Yaskawa INFORM job: A_ROOF_UPPER_0614_2_PAINT_56.JBI

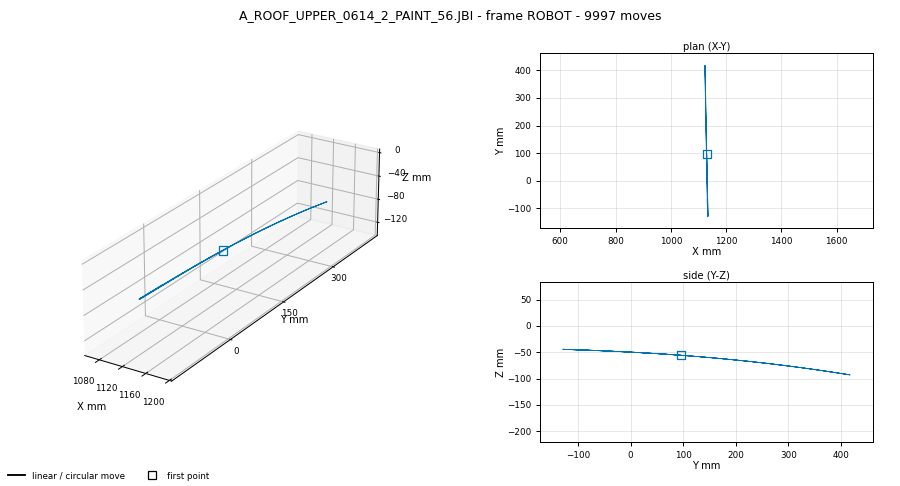
[picture p0: tool path of A_ROOF_UPPER_0614_2_PAINT_56.JBI in frame ROBOT, 9997 of 9997 moves have a stored position in this frame; points joined in program order, loops and branches not executed]
/JOB
//NAME A_ROOF_UPPER_0614_2_PAINT56
//POS
///NPOS 9997,0,0,0,0,0
///TOOL 1
///USER 0
///POSTYPE ROBOT
///RECTAN
///RCONF 1,0,0,0,0,0,0,0,0,0,0,0,0,0,0,0,0,0,0,0,0,0,0,0
C00000=1130.429,96.050,-55.597,-179.993,7.913,149.501
C00001=1130.433,95.801,-55.579,-179.995,7.908,149.501
C00002=1130.438,95.552,-55.561,-179.997,7.904,149.500
C00003=1130.443,95.303,-55.543,-179.999,7.901,149.500
C00004=1130.448,95.054,-55.525,180.000,7.897,149.500
C00005=1130.453,94.805,-55.507,179.998,7.893,149.499
C00006=1130.457,94.555,-55.488,179.996,7.888,149.499
C00007=1130.463,94.305,-55.470,179.994,7.884,149.499
C00008=1130.468,94.056,-55.452,179.993,7.881,149.498
C00009=1130.473,93.807,-55.434,179.991,7.877,149.498
C00010=1130.478,93.558,-55.416,179.989,7.873,149.497
C00011=1130.483,93.308,-55.398,179.987,7.869,149.497
C00012=1130.488,93.059,-55.380,179.986,7.865,149.497
C00013=1130.493,92.810,-55.362,179.984,7.861,149.496
C00014=1130.497,92.560,-55.344,179.982,7.857,149.496
C00015=1130.502,92.311,-55.326,179.980,7.853,149.495
C00016=1130.507,92.062,-55.308,179.979,7.849,149.495
C00017=1130.512,91.813,-55.290,179.977,7.845,149.495
C00018=1130.517,91.564,-55.272,179.976,7.841,149.494
C00019=1130.521,91.314,-55.254,179.974,7.837,149.494
C00020=1130.526,91.065,-55.236,179.972,7.833,149.493
C00021=1130.532,90.815,-55.218,179.971,7.830,149.493
C00022=1130.536,90.566,-55.200,179.970,7.825,149.492
C00023=1130.541,90.317,-55.182,179.968,7.821,149.492
C00024=1130.545,90.102,-55.167,179.967,7.819,149.492
C00025=1130.549,89.887,-55.151,179.965,7.815,149.491
C00026=1130.553,89.672,-55.137,179.964,7.812,149.491
C00027=1130.558,89.457,-55.121,179.963,7.808,149.490
C00028=1130.562,89.242,-55.105,179.962,7.805,149.490
C00029=1130.567,89.027,-55.090,179.960,7.801,149.489
C00030=1130.570,88.811,-55.075,179.959,7.798,149.489
C00031=1130.575,88.596,-55.060,179.958,7.795,149.489
C00032=1130.579,88.347,-55.042,179.956,7.791,149.488
C00033=1130.585,88.097,-55.024,179.955,7.787,149.488
C00034=1130.590,87.848,-55.006,179.953,7.783,149.487
C00035=1130.594,87.599,-54.989,179.952,7.779,149.487
C00036=1130.599,87.350,-54.971,179.950,7.775,149.486
C00037=1130.604,87.100,-54.954,179.949,7.771,149.486
C00038=1130.609,86.851,-54.936,179.947,7.767,149.485
C00039=1130.614,86.602,-54.918,179.946,7.764,149.485
C00040=1130.619,86.352,-54.900,179.945,7.760,149.485
C00041=1130.623,86.103,-54.883,179.944,7.756,149.484
C00042=1130.628,85.854,-54.865,179.942,7.752,149.483
C00043=1130.633,85.604,-54.848,179.940,7.748,149.483
C00044=1130.638,85.355,-54.830,179.939,7.744,149.483
C00045=1130.643,85.105,-54.813,179.938,7.740,149.482
C00046=1130.648,84.856,-54.795,179.937,7.737,149.482
C00047=1130.653,84.608,-54.778,179.935,7.733,149.481
C00048=1130.658,84.358,-54.760,179.934,7.728,149.480
C00049=1130.663,84.109,-54.742,179.933,7.725,149.480
C00050=1130.668,83.859,-54.725,179.931,7.721,149.480
C00051=1130.673,83.610,-54.708,179.930,7.717,149.479
C00052=1130.678,83.361,-54.690,179.929,7.713,149.479
C00053=1130.683,83.111,-54.672,179.928,7.710,149.478
C00054=1130.688,82.862,-54.655,179.927,7.706,149.477
C00055=1130.692,82.613,-54.638,179.925,7.702,149.477
C00056=1130.697,82.363,-54.621,179.925,7.698,149.476
C00057=1130.702,82.114,-54.603,179.923,7.694,149.476
C00058=1130.707,81.864,-54.586,179.922,7.690,149.475
C00059=1130.712,81.615,-54.568,179.921,7.687,149.475
C00060=1130.717,81.366,-54.551,179.920,7.683,149.474
C00061=1130.722,81.117,-54.534,179.919,7.680,149.474
C00062=1130.727,80.867,-54.516,179.918,7.675,149.473
C00063=1130.732,80.618,-54.499,179.916,7.672,149.473
C00064=1130.736,80.369,-54.482,179.916,7.668,149.472
C00065=1130.741,80.119,-54.464,179.914,7.664,149.472
C00066=1130.746,79.870,-54.446,179.913,7.661,149.471
C00067=1130.751,79.620,-54.430,179.912,7.657,149.471
C00068=1130.757,79.371,-54.413,179.911,7.653,149.470
C00069=1130.762,79.122,-54.395,179.910,7.649,149.470
C00070=1130.766,78.872,-54.378,179.909,7.645,149.469
C00071=1130.771,78.623,-54.361,179.908,7.642,149.469
C00072=1130.776,78.373,-54.343,179.907,7.638,149.468
C00073=1130.781,78.124,-54.326,179.906,7.634,149.467
C00074=1130.786,77.874,-54.309,179.905,7.631,149.467
C00075=1130.791,77.626,-54.292,179.903,7.627,149.466
C00076=1130.796,77.376,-54.275,179.903,7.624,149.466
C00077=1130.801,77.126,-54.257,179.902,7.619,149.465
C00078=1130.805,76.878,-54.240,179.901,7.616,149.465
C00079=1130.810,76.628,-54.223,179.900,7.612,149.464
C00080=1130.819,76.209,-54.195,179.897,7.606,149.463
C00081=1130.827,75.790,-54.166,179.895,7.599,149.463
C00082=1130.835,75.371,-54.137,179.892,7.592,149.462
C00083=1130.844,74.952,-54.108,179.890,7.586,149.461
C00084=1130.849,74.703,-54.092,179.889,7.582,149.460
C00085=1130.854,74.454,-54.074,179.887,7.578,149.460
C00086=1130.858,74.204,-54.057,179.886,7.574,149.460
C00087=1130.863,73.954,-54.040,179.885,7.570,149.459
C00088=1130.868,73.705,-54.023,179.883,7.566,149.458
C00089=1130.873,73.456,-54.007,179.881,7.562,149.458
C00090=1130.878,73.206,-53.990,179.880,7.558,149.458
C00091=1130.883,72.957,-53.973,179.879,7.554,149.457
C00092=1130.888,72.707,-53.956,179.877,7.550,149.457
C00093=1130.893,72.459,-53.939,179.876,7.546,149.456
C00094=1130.898,72.209,-53.922,179.874,7.542,149.456
C00095=1130.902,71.960,-53.905,179.873,7.538,149.455
C00096=1130.908,71.711,-53.888,179.871,7.534,149.455
C00097=1130.913,71.461,-53.871,179.870,7.530,149.454
C00098=1130.917,71.212,-53.855,179.868,7.526,149.454
C00099=1130.922,70.962,-53.837,179.867,7.522,149.453
C00100=1130.928,70.713,-53.821,179.865,7.518,149.453
C00101=1130.933,70.463,-53.804,179.864,7.514,149.452
C00102=1130.937,70.214,-53.787,179.862,7.510,149.452
C00103=1130.942,69.965,-53.771,179.861,7.506,149.451
C00104=1130.968,68.716,-53.685,-179.718,6.654,149.139
C00105=1130.972,68.467,-53.668,-179.720,6.653,149.139
C00106=1130.977,68.217,-53.652,-179.723,6.652,149.139
C00107=1130.982,67.969,-53.636,-179.726,6.650,149.140
C00108=1130.986,67.718,-53.620,-179.728,6.648,149.140
C00109=1130.992,67.469,-53.603,-179.731,6.648,149.141
C00110=1130.997,67.220,-53.586,-179.734,6.646,149.141
C00111=1131.002,66.970,-53.570,-179.736,6.645,149.142
C00112=1131.007,66.721,-53.554,-179.739,6.643,149.142
C00113=1131.011,66.471,-53.537,-179.741,6.642,149.143
C00114=1131.017,66.222,-53.521,-179.745,6.641,149.143
C00115=1131.022,65.972,-53.504,-179.747,6.639,149.144
C00116=1131.027,65.724,-53.488,-179.750,6.638,149.144
C00117=1131.032,65.473,-53.472,-179.752,6.637,149.145
C00118=1131.037,65.225,-53.456,-179.756,6.636,149.145
C00119=1131.041,64.975,-53.439,-179.758,6.634,149.146
C00120=1131.047,64.726,-53.423,-179.760,6.633,149.146
C00121=1131.051,64.476,-53.407,-179.763,6.631,149.147
C00122=1131.056,64.227,-53.391,-179.766,6.630,149.147
C00123=1131.061,63.977,-53.374,-179.769,6.629,149.148
C00124=1131.066,63.728,-53.359,-179.771,6.628,149.148
C00125=1131.071,63.478,-53.342,-179.774,6.626,149.149
C00126=1131.077,63.229,-53.325,-179.777,6.624,149.149
C00127=1131.081,62.979,-53.309,-179.779,6.624,149.150
C00128=1131.086,62.730,-53.293,-179.782,6.622,149.150
C00129=1131.091,62.480,-53.277,-179.785,6.621,149.151
C00130=1131.096,62.232,-53.261,-179.787,6.620,149.151
C00131=1131.101,61.981,-53.245,-179.790,6.619,149.152
C00132=1131.106,61.733,-53.229,-179.793,6.617,149.152
C00133=1131.112,61.483,-53.213,-179.795,6.616,149.153
C00134=1131.116,61.234,-53.196,-179.798,6.614,149.153
C00135=1131.121,60.984,-53.181,-179.801,6.613,149.154
C00136=1131.126,60.734,-53.165,-179.803,6.612,149.154
C00137=1131.131,60.486,-53.148,-179.806,6.611,149.155
C00138=1131.136,60.235,-53.133,-179.809,6.609,149.155
C00139=1131.141,59.987,-53.116,-179.811,6.608,149.155
C00140=1131.147,59.737,-53.101,-179.814,6.607,149.156
C00141=1131.151,59.487,-53.085,-179.817,6.605,149.157
C00142=1131.156,59.238,-53.068,-179.819,6.605,149.157
C00143=1131.161,58.988,-53.052,-179.822,6.603,149.157
C00144=1131.166,58.739,-53.036,-179.825,6.602,149.158
C00145=1131.172,58.490,-53.021,-179.827,6.601,149.159
C00146=1131.176,58.240,-53.005,-179.830,6.599,149.159
C00147=1131.181,57.992,-52.989,-179.833,6.598,149.159
C00148=1131.186,57.741,-52.973,-179.836,6.597,149.160
C00149=1131.191,57.492,-52.957,-179.838,6.595,149.161
C00150=1131.196,57.243,-52.942,-179.841,6.594,149.161
C00151=1131.201,56.993,-52.925,-179.843,6.593,149.161
C00152=1131.206,56.744,-52.909,-179.847,6.592,149.162
C00153=1131.212,56.494,-52.894,-179.849,6.590,149.163
C00154=1131.216,56.245,-52.877,-179.851,6.589,149.163
C00155=1131.221,55.995,-52.862,-179.854,6.588,149.163
C00156=1131.226,55.746,-52.847,-179.857,6.586,149.164
C00157=1131.231,55.496,-52.831,-179.860,6.586,149.165
C00158=1131.236,55.247,-52.815,-179.862,6.584,149.165
C00159=1131.241,54.998,-52.799,-179.865,6.582,149.165
C00160=1131.246,54.748,-52.783,-179.868,6.582,149.166
C00161=1131.252,54.499,-52.767,-179.870,6.580,149.167
C00162=1131.256,54.249,-52.752,-179.873,6.579,149.167
C00163=1131.261,53.999,-52.736,-179.875,6.578,149.167
C00164=1131.266,53.751,-52.720,-179.879,6.576,149.168
C00165=1131.272,53.481,-52.704,-179.881,6.575,149.168
C00166=1131.277,53.213,-52.687,-179.884,6.574,149.169
C00167=1131.283,52.944,-52.670,-179.887,6.573,149.170
C00168=1131.289,52.676,-52.653,-179.890,6.571,149.170
C00169=1131.293,52.426,-52.637,-179.893,6.570,149.171
C00170=1131.298,52.177,-52.622,-179.895,6.569,149.171
C00171=1131.303,51.927,-52.606,-179.898,6.567,149.172
C00172=1131.308,51.677,-52.590,-179.901,6.566,149.172
C00173=1131.313,51.428,-52.575,-179.903,6.565,149.173
C00174=1131.318,51.179,-52.560,-179.906,6.564,149.173
C00175=1131.324,50.929,-52.544,-179.908,6.563,149.174
C00176=1131.328,50.680,-52.529,-179.911,6.562,149.174
C00177=1131.333,50.430,-52.513,-179.914,6.560,149.175
C00178=1131.338,50.181,-52.497,-179.916,6.559,149.175
C00179=1131.344,49.932,-52.481,-179.919,6.557,149.176
C00180=1131.348,49.682,-52.466,-179.922,6.557,149.176
C00181=1131.353,49.433,-52.450,-179.924,6.555,149.177
C00182=1131.359,49.183,-52.435,-179.927,6.554,149.177
C00183=1131.363,48.934,-52.420,-179.929,6.553,149.178
C00184=1131.369,48.684,-52.405,-179.933,6.552,149.178
C00185=1131.373,48.434,-52.389,-179.935,6.551,149.179
C00186=1131.378,48.185,-52.374,-179.937,6.549,149.179
C00187=1131.384,47.936,-52.358,-179.941,6.548,149.180
C00188=1131.388,47.687,-52.343,-179.943,6.547,149.180
C00189=1131.394,47.437,-52.328,-179.946,6.546,149.181
C00190=1131.398,47.187,-52.312,-179.948,6.545,149.181
C00191=1131.403,46.938,-52.297,-179.951,6.543,149.182
C00192=1131.408,46.689,-52.281,-179.953,6.543,149.182
C00193=1131.414,46.439,-52.266,-179.956,6.541,149.183
C00194=1131.419,46.190,-52.251,-179.959,6.539,149.183
C00195=1131.424,45.939,-52.235,-179.961,6.539,149.184
C00196=1131.428,45.690,-52.220,-179.964,6.537,149.184
C00197=1131.434,45.441,-52.205,-179.966,6.536,149.185
C00198=1131.438,45.192,-52.190,-179.970,6.535,149.185
C00199=1131.444,44.942,-52.174,-179.972,6.534,149.186
C00200=1131.449,44.692,-52.159,-179.974,6.533,149.186
C00201=1131.454,44.443,-52.144,-179.977,6.531,149.187
C00202=1131.459,44.193,-52.128,-179.980,6.531,149.187
C00203=1131.463,43.944,-52.113,-179.983,6.529,149.188
C00204=1131.469,43.695,-52.098,-179.985,6.528,149.188
C00205=1131.474,43.445,-52.083,-179.988,6.527,149.189
C00206=1131.479,43.196,-52.068,-179.990,6.526,149.189
C00207=1131.484,42.947,-52.053,-179.993,6.525,149.190
C00208=1131.489,42.697,-52.038,-179.995,6.524,149.190
C00209=1131.494,42.447,-52.023,-179.998,6.522,149.191
C00210=1131.499,42.198,-52.007,179.999,6.522,149.191
C00211=1131.504,41.949,-51.992,179.997,6.520,149.192
C00212=1131.509,41.698,-51.977,179.994,6.518,149.192
C00213=1131.514,41.449,-51.962,179.991,6.518,149.193
C00214=1131.519,41.200,-51.947,179.989,6.516,149.193
C00215=1131.524,40.950,-51.932,179.986,6.516,149.194
C00216=1131.530,40.701,-51.917,179.983,6.514,149.195
C00217=1131.534,40.452,-51.902,179.981,6.513,149.195
C00218=1131.539,40.202,-51.887,179.978,6.512,149.196
C00219=1131.545,39.952,-51.872,179.976,6.511,149.196
C00220=1131.550,39.703,-51.858,179.973,6.510,149.197
C00221=1131.555,39.453,-51.842,179.971,6.509,149.197
C00222=1131.560,39.204,-51.827,179.968,6.507,149.198
C00223=1131.565,38.954,-51.813,179.965,6.507,149.198
C00224=1131.570,38.705,-51.797,179.962,6.505,149.199
C00225=1131.575,38.455,-51.783,179.960,6.504,149.199
C00226=1131.580,38.206,-51.767,179.957,6.503,149.200
C00227=1131.585,37.956,-51.753,179.955,6.502,149.200
C00228=1131.590,37.707,-51.738,179.952,6.501,149.201
C00229=1131.596,37.457,-51.723,179.950,6.500,149.201
C00230=1131.600,37.208,-51.708,179.947,6.499,149.202
C00231=1131.606,36.958,-51.693,179.945,6.498,149.202
C00232=1131.611,36.709,-51.678,179.942,6.496,149.203
C00233=1131.615,36.459,-51.664,179.939,6.496,149.203
C00234=1131.621,36.210,-51.648,179.936,6.494,149.204
C00235=1131.626,35.960,-51.634,179.934,6.493,149.204
C00236=1131.630,35.711,-51.619,179.931,6.492,149.205
C00237=1131.636,35.461,-51.604,179.929,6.491,149.205
C00238=1131.641,35.212,-51.589,179.926,6.490,149.206
C00239=1131.646,34.962,-51.575,179.924,6.489,149.206
C00240=1131.650,34.713,-51.560,179.921,6.488,149.207
C00241=1131.656,34.463,-51.545,179.918,6.487,149.207
C00242=1131.661,34.213,-51.531,179.916,6.485,149.208
C00243=1131.666,33.964,-51.516,179.913,6.485,149.209
C00244=1131.671,33.715,-51.502,179.910,6.483,149.209
C00245=1131.676,33.465,-51.487,179.908,6.482,149.209
C00246=1131.681,33.215,-51.472,179.905,6.481,149.210
C00247=1131.686,32.966,-51.457,179.903,6.480,149.211
C00248=1131.691,32.716,-51.443,179.900,6.479,149.211
C00249=1131.697,32.467,-51.428,179.898,6.478,149.212
C00250=1131.702,32.218,-51.414,179.894,6.477,149.212
C00251=1131.707,31.968,-51.399,179.892,6.476,149.213
C00252=1131.711,31.719,-51.384,179.890,6.474,149.213
C00253=1131.717,31.469,-51.370,179.887,6.474,149.214
C00254=1131.722,31.219,-51.355,179.884,6.472,149.214
C00255=1131.727,30.970,-51.340,179.882,6.471,149.215
C00256=1131.732,30.720,-51.326,179.879,6.470,149.215
C00257=1131.737,30.471,-51.312,179.877,6.469,149.216
C00258=1131.742,30.221,-51.297,179.874,6.468,149.216
C00259=1131.748,29.972,-51.282,179.872,6.467,149.217
C00260=1131.753,29.722,-51.268,179.869,6.466,149.217
C00261=1131.758,29.473,-51.254,179.866,6.465,149.218
C00262=1131.762,29.223,-51.239,179.864,6.464,149.218
C00263=1131.767,28.973,-51.225,179.861,6.463,149.219
C00264=1131.772,28.724,-51.210,179.859,6.462,149.219
C00265=1131.777,28.475,-51.196,179.856,6.460,149.220
C00266=1131.783,28.225,-51.181,179.854,6.459,149.220
C00267=1131.788,27.975,-51.167,179.851,6.459,149.221
C00268=1131.793,27.726,-51.153,179.848,6.457,149.221
C00269=1131.798,27.457,-51.137,179.845,6.456,149.222
C00270=1131.804,27.188,-51.121,179.843,6.455,149.223
C00271=1131.809,26.919,-51.106,179.840,6.454,149.223
C00272=1131.815,26.650,-51.090,179.837,6.453,149.224
C00273=1131.820,26.401,-51.076,179.835,6.452,149.224
C00274=1131.825,26.151,-51.062,179.832,6.451,149.225
C00275=1131.830,25.901,-51.048,179.829,6.450,149.225
C00276=1131.835,25.652,-51.033,179.827,6.449,149.226
C00277=1131.840,25.402,-51.019,179.824,6.448,149.226
C00278=1131.846,25.153,-51.005,179.822,6.447,149.227
C00279=1131.851,24.903,-50.991,179.819,6.446,149.227
C00280=1131.856,24.653,-50.977,179.816,6.445,149.228
C00281=1131.861,24.404,-50.962,179.814,6.444,149.229
C00282=1131.866,24.155,-50.948,179.811,6.442,149.229
C00283=1131.871,23.905,-50.934,179.809,6.441,149.229
C00284=1131.876,23.655,-50.920,179.806,6.441,149.230
C00285=1131.881,23.406,-50.906,179.804,6.439,149.231
C00286=1131.886,23.156,-50.891,179.801,6.439,149.231
C00287=1131.892,22.907,-50.877,179.798,6.437,149.232
C00288=1131.896,22.657,-50.863,179.796,6.437,149.232
C00289=1131.901,22.407,-50.849,179.794,6.436,149.233
C00290=1131.906,22.158,-50.835,179.791,6.434,149.233
C00291=1131.912,21.909,-50.821,179.788,6.434,149.234
C00292=1131.917,21.659,-50.806,179.786,6.432,149.234
C00293=1131.922,21.409,-50.792,179.783,6.432,149.235
C00294=1131.927,21.160,-50.778,179.781,6.431,149.235
C00295=1131.932,20.911,-50.764,179.778,6.429,149.236
C00296=1131.937,20.661,-50.750,179.775,6.429,149.237
C00297=1131.942,20.411,-50.737,179.773,6.427,149.237
C00298=1131.947,20.162,-50.723,179.771,6.426,149.237
C00299=1131.952,19.912,-50.708,179.768,6.426,149.238
C00300=1131.957,19.662,-50.694,179.765,6.424,149.239
C00301=1131.963,19.413,-50.680,179.763,6.423,149.239
C00302=1131.968,19.164,-50.666,179.760,6.422,149.239
C00303=1131.973,18.914,-50.652,179.757,6.421,149.240
C00304=1131.979,18.664,-50.639,179.755,6.421,149.241
C00305=1131.983,18.415,-50.625,179.753,6.419,149.241
C00306=1131.988,18.165,-50.611,179.750,6.419,149.242
C00307=1131.993,17.916,-50.597,179.748,6.418,149.242
C00308=1131.998,17.666,-50.582,179.745,6.416,149.243
C00309=1132.004,17.416,-50.569,179.742,6.416,149.243
C00310=1132.009,17.167,-50.555,179.740,6.415,149.244
C00311=1132.013,16.918,-50.541,179.737,6.413,149.244
C00312=1132.018,16.668,-50.527,179.735,6.413,149.245
C00313=1132.024,16.418,-50.514,179.732,6.411,149.245
C00314=1132.029,16.169,-50.499,179.730,6.411,149.246
C00315=1132.034,15.919,-50.485,179.727,6.410,149.247
C00316=1132.039,15.670,-50.473,179.724,6.408,149.247
C00317=1132.044,15.420,-50.458,179.722,6.408,149.248
C00318=1132.049,15.170,-50.444,179.719,6.407,149.248
C00319=1132.055,14.921,-50.430,179.717,6.406,149.249
C00320=1132.060,14.671,-50.417,179.715,6.405,149.249
C00321=1132.065,14.422,-50.403,179.712,6.404,149.250
C00322=1132.070,14.173,-50.389,179.709,6.403,149.250
C00323=1132.075,13.922,-50.375,179.707,6.402,149.251
C00324=1132.081,13.673,-50.361,179.705,6.401,149.251
C00325=1132.085,13.423,-50.349,179.702,6.400,149.252
C00326=1132.091,13.174,-50.335,179.699,6.399,149.252
C00327=1132.096,12.924,-50.320,179.697,6.398,149.253
C00328=1132.101,12.675,-50.308,179.694,6.397,149.253
C00329=1132.106,12.425,-50.293,179.692,6.396,149.254
C00330=1132.111,12.175,-50.280,179.690,6.395,149.254
C00331=1132.116,11.926,-50.266,179.686,6.394,149.255
C00332=1132.121,11.677,-50.252,179.684,6.393,149.256
C00333=1132.127,11.427,-50.239,179.682,6.393,149.256
C00334=1132.131,11.177,-50.225,179.679,6.391,149.257
C00335=1132.137,10.928,-50.212,179.677,6.391,149.257
C00336=1132.142,10.678,-50.198,179.674,6.390,149.258
C00337=1132.147,10.429,-50.185,179.671,6.389,149.258
C00338=1132.152,10.179,-50.171,179.669,6.388,149.259
C00339=1132.157,9.929,-50.158,179.667,6.387,149.259
C00340=1132.162,9.680,-50.144,179.663,6.386,149.260
C00341=1132.167,9.430,-50.131,179.661,6.385,149.260
C00342=1132.173,9.181,-50.117,179.659,6.384,149.261
C00343=1132.177,8.931,-50.104,179.656,6.384,149.262
C00344=1132.183,8.682,-50.090,179.654,6.382,149.262
C00345=1132.188,8.432,-50.076,179.652,6.381,149.262
C00346=1132.193,8.183,-50.063,179.649,6.381,149.263
C00347=1132.198,7.933,-50.049,179.646,6.379,149.264
C00348=1132.203,7.683,-50.037,179.644,6.379,149.264
C00349=1132.208,7.433,-50.023,179.642,6.378,149.265
C00350=1132.214,7.184,-50.009,179.639,6.376,149.265
C00351=1132.218,6.934,-49.996,179.636,6.376,149.266
C00352=1132.224,6.685,-49.982,179.634,6.375,149.266
C00353=1132.228,6.435,-49.969,179.632,6.374,149.267
C00354=1132.234,6.186,-49.956,179.629,6.373,149.267
C00355=1132.239,5.936,-49.943,179.627,6.372,149.268
C00356=1132.244,5.686,-49.929,179.624,6.372,149.268
C00357=1132.249,5.437,-49.916,179.621,6.370,149.269
C00358=1132.255,5.187,-49.903,179.619,6.369,149.269
C00359=1132.260,4.937,-49.889,179.616,6.369,149.270
C00360=1132.265,4.688,-49.876,179.614,6.368,149.271
C00361=1132.270,4.438,-49.862,179.611,6.366,149.271
C00362=1132.275,4.188,-49.849,179.609,6.366,149.272
C00363=1132.281,3.939,-49.836,179.606,6.365,149.272
C00364=1132.286,3.690,-49.823,179.604,6.364,149.273
C00365=1132.291,3.440,-49.809,179.601,6.363,149.273
C00366=1132.296,3.190,-49.797,179.599,6.362,149.274
C00367=1132.300,2.941,-49.783,179.597,6.362,149.274
C00368=1132.306,2.691,-49.770,179.593,6.360,149.275
C00369=1132.311,2.441,-49.757,179.591,6.360,149.275
C00370=1132.317,2.192,-49.744,179.589,6.359,149.276
C00371=1132.321,1.943,-49.730,179.586,6.358,149.277
C00372=1132.327,1.693,-49.717,179.584,6.357,149.277
C00373=1132.332,1.424,-49.704,179.581,6.356,149.277
C00374=1132.338,1.154,-49.689,179.579,6.356,149.278
C00375=1132.343,0.884,-49.674,179.576,6.354,149.279
C00376=1132.348,0.615,-49.661,179.573,6.354,149.279
C00377=1132.354,0.365,-49.647,179.571,6.352,149.280
C00378=1132.359,0.116,-49.635,179.568,6.352,149.280
C00379=1132.364,-0.134,-49.621,179.566,6.351,149.281
C00380=1132.369,-0.383,-49.608,179.564,6.350,149.281
C00381=1132.375,-0.633,-49.595,179.560,6.349,149.282
C00382=1132.380,-0.883,-49.582,179.558,6.348,149.283
C00383=1132.385,-1.132,-49.569,179.556,6.347,149.283
C00384=1132.390,-1.382,-49.557,179.553,6.347,149.284
C00385=1132.395,-1.632,-49.543,179.551,6.346,149.284
C00386=1132.400,-1.881,-49.530,179.548,6.344,149.285
C00387=1132.406,-2.131,-49.518,179.546,6.343,149.285
C00388=1132.411,-2.380,-49.504,179.544,6.343,149.286
C00389=1132.416,-2.630,-49.491,179.541,6.342,149.286
C00390=1132.421,-2.879,-49.478,179.539,6.341,149.287
C00391=1132.426,-3.129,-49.465,179.536,6.340,149.287
C00392=1132.431,-3.379,-49.452,179.534,6.339,149.288
C00393=1132.436,-3.628,-49.440,179.532,6.339,149.288
C00394=1132.442,-3.878,-49.426,179.528,6.337,149.289
C00395=1132.447,-4.128,-49.413,179.526,6.337,149.289
C00396=1132.452,-4.377,-49.401,179.524,6.336,149.290
C00397=1132.458,-4.627,-49.388,179.521,6.335,149.291
C00398=1132.462,-4.877,-49.375,179.519,6.335,149.291
C00399=1132.467,-5.126,-49.362,179.516,6.333,149.292
C00400=1132.472,-5.375,-49.349,179.514,6.333,149.292
C00401=1132.478,-5.626,-49.336,179.511,6.332,149.293
C00402=1132.483,-5.875,-49.323,179.509,6.331,149.293
C00403=1132.488,-6.125,-49.311,179.507,6.331,149.294
C00404=1132.493,-6.374,-49.299,179.504,6.329,149.294
C00405=1132.499,-6.624,-49.285,179.502,6.328,149.295
C00406=1132.504,-6.874,-49.273,179.499,6.328,149.296
C00407=1132.509,-7.123,-49.260,179.497,6.327,149.296
C00408=1132.514,-7.372,-49.247,179.495,6.326,149.296
C00409=1132.519,-7.623,-49.234,179.491,6.325,149.297
C00410=1132.524,-7.872,-49.221,179.489,6.324,149.298
C00411=1132.529,-8.121,-49.209,179.487,6.323,149.298
C00412=1132.535,-8.371,-49.196,179.484,6.323,149.299
C00413=1132.540,-8.621,-49.184,179.482,6.322,149.299
C00414=1132.545,-8.871,-49.171,179.479,6.321,149.300
C00415=1132.550,-9.120,-49.158,179.477,6.320,149.300
C00416=1132.556,-9.370,-49.145,179.475,6.319,149.301
C00417=1132.561,-9.619,-49.133,179.472,6.319,149.301
C00418=1132.565,-9.869,-49.120,179.470,6.318,149.302
C00419=1132.571,-10.119,-49.108,179.468,6.317,149.303
C00420=1132.576,-10.368,-49.095,179.465,6.316,149.303
C00421=1132.582,-10.618,-49.082,179.463,6.315,149.303
C00422=1132.587,-10.867,-49.070,179.460,6.315,149.304
C00423=1132.592,-11.118,-49.057,179.458,6.314,149.305
C00424=1132.597,-11.367,-49.045,179.456,6.313,149.305
C00425=1132.602,-11.616,-49.032,179.453,6.313,149.306
C00426=1132.607,-11.866,-49.020,179.450,6.311,149.306
C00427=1132.612,-12.116,-49.008,179.448,6.310,149.307
C00428=1132.617,-12.365,-48.995,179.445,6.310,149.307
C00429=1132.622,-12.615,-48.982,179.443,6.309,149.308
C00430=1132.628,-12.865,-48.969,179.441,6.308,149.308
C00431=1132.633,-13.115,-48.957,179.438,6.308,149.309
C00432=1132.638,-13.364,-48.944,179.435,6.306,149.310
C00433=1132.644,-13.613,-48.932,179.433,6.306,149.310
C00434=1132.649,-13.863,-48.920,179.431,6.305,149.311
C00435=1132.654,-14.112,-48.907,179.428,6.304,149.311
C00436=1132.659,-14.362,-48.894,179.426,6.304,149.312
C00437=1132.664,-14.612,-48.882,179.424,6.303,149.312
C00438=1132.669,-14.862,-48.870,179.421,6.302,149.313
C00439=1132.674,-15.111,-48.857,179.419,6.301,149.313
C00440=1132.680,-15.361,-48.845,179.416,6.300,149.314
C00441=1132.685,-15.610,-48.833,179.414,6.300,149.314
C00442=1132.690,-15.860,-48.820,179.412,6.299,149.315
C00443=1132.695,-16.110,-48.808,179.409,6.298,149.315
C00444=1132.700,-16.360,-48.795,179.407,6.298,149.316
C00445=1132.705,-16.609,-48.783,179.405,6.297,149.317
C00446=1132.710,-16.859,-48.771,179.402,6.295,149.317
C00447=1132.716,-17.109,-48.759,179.399,6.295,149.318
C00448=1132.721,-17.358,-48.746,179.397,6.294,149.318
C00449=1132.726,-17.607,-48.734,179.395,6.293,149.319
C00450=1132.732,-17.857,-48.722,179.392,6.293,149.319
C00451=1132.737,-18.107,-48.709,179.390,6.292,149.320
C00452=1132.742,-18.357,-48.697,179.388,6.291,149.320
C00453=1132.747,-18.606,-48.685,179.386,6.290,149.321
C00454=1132.753,-18.856,-48.673,179.382,6.289,149.321
C00455=1132.758,-19.105,-48.660,179.380,6.288,149.322
C00456=1132.763,-19.355,-48.648,179.378,6.288,149.322
C00457=1132.768,-19.604,-48.636,179.375,6.287,149.323
C00458=1132.774,-19.854,-48.624,179.373,6.286,149.324
C00459=1132.778,-20.103,-48.612,179.371,6.286,149.324
C00460=1132.783,-20.354,-48.600,179.368,6.285,149.325
C00461=1132.788,-20.604,-48.588,179.366,6.284,149.325
C00462=1132.794,-20.853,-48.575,179.364,6.284,149.326
C00463=1132.799,-21.103,-48.563,179.361,6.283,149.326
C00464=1132.804,-21.352,-48.551,179.358,6.282,149.327
C00465=1132.810,-21.602,-48.539,179.356,6.281,149.327
C00466=1132.815,-21.852,-48.526,179.354,6.281,149.328
C00467=1132.820,-22.102,-48.514,179.351,6.280,149.328
C00468=1132.826,-22.352,-48.502,179.349,6.279,149.329
C00469=1132.830,-22.601,-48.490,179.347,6.278,149.329
C00470=1132.835,-22.851,-48.479,179.344,6.278,149.330
C00471=1132.840,-23.100,-48.466,179.342,6.277,149.331
C00472=1132.846,-23.350,-48.454,179.340,6.276,149.331
C00473=1132.851,-23.600,-48.442,179.337,6.275,149.332
C00474=1132.856,-23.849,-48.430,179.335,6.274,149.332
C00475=1132.862,-24.098,-48.419,179.332,6.273,149.333
C00476=1132.867,-24.348,-48.407,179.330,6.273,149.333
C00477=1132.873,-24.618,-48.394,179.328,6.272,149.334
C00478=1132.879,-24.889,-48.380,179.325,6.272,149.335
C00479=1132.884,-25.159,-48.368,179.322,6.270,149.335
C00480=1132.890,-25.429,-48.355,179.319,6.270,149.336
C00481=1132.895,-25.678,-48.342,179.317,6.269,149.336
C00482=1132.900,-25.928,-48.331,179.315,6.268,149.337
C00483=1132.905,-26.178,-48.319,179.313,6.268,149.337
C00484=1132.910,-26.428,-48.307,179.310,6.267,149.338
C00485=1132.916,-26.677,-48.294,179.308,6.266,149.338
C00486=1132.920,-26.927,-48.283,179.306,6.266,149.339
C00487=1132.926,-27.177,-48.271,179.303,6.265,149.339
C00488=1132.931,-27.427,-48.259,179.301,6.264,149.340
C00489=1132.937,-27.675,-48.247,179.299,6.264,149.340
C00490=1132.942,-27.925,-48.236,179.296,6.263,149.341
C00491=1132.947,-28.175,-48.224,179.293,6.262,149.342
C00492=1132.952,-28.425,-48.212,179.291,6.261,149.342
C00493=1132.958,-28.675,-48.200,179.289,6.260,149.343
C00494=1132.962,-28.924,-48.188,179.286,6.260,149.343
C00495=1132.968,-29.174,-48.176,179.284,6.259,149.344
C00496=1132.973,-29.424,-48.164,179.282,6.258,149.344
C00497=1132.978,-29.673,-48.153,179.279,6.258,149.345
C00498=1132.983,-29.923,-48.141,179.277,6.257,149.345
C00499=1132.989,-30.172,-48.130,179.275,6.256,149.346
C00500=1132.994,-30.421,-48.118,179.272,6.256,149.347
C00501=1132.999,-30.671,-48.106,179.270,6.255,149.347
C00502=1133.004,-30.921,-48.094,179.268,6.254,149.348
C00503=1133.009,-31.171,-48.083,179.266,6.253,149.348
C00504=1133.015,-31.421,-48.071,179.263,6.253,149.349
C00505=1133.020,-31.671,-48.059,179.261,6.252,149.349
C00506=1133.025,-31.920,-48.048,179.259,6.251,149.350
C00507=1133.031,-32.170,-48.036,179.256,6.251,149.350
C00508=1133.036,-32.419,-48.024,179.254,6.250,149.351
C00509=1133.041,-32.669,-48.013,179.252,6.249,149.351
C00510=1133.046,-32.919,-48.001,179.249,6.249,149.352
C00511=1133.051,-33.169,-47.990,179.247,6.248,149.352
C00512=1133.056,-33.418,-47.977,179.245,6.248,149.353
C00513=1133.062,-33.667,-47.966,179.242,6.247,149.353
C00514=1133.067,-33.917,-47.954,179.240,6.246,149.354
C00515=1133.072,-34.167,-47.942,179.238,6.246,149.355
C00516=1133.077,-34.416,-47.931,179.235,6.244,149.355
C00517=1133.082,-34.666,-47.919,179.232,6.244,149.356
C00518=1133.088,-34.916,-47.908,179.230,6.243,149.356
C00519=1133.093,-35.165,-47.896,179.228,6.242,149.357
C00520=1133.099,-35.415,-47.885,179.225,6.241,149.357
C00521=1133.104,-35.665,-47.874,179.223,6.241,149.358
C00522=1133.109,-35.915,-47.862,179.221,6.240,149.358
C00523=1133.114,-36.164,-47.851,179.218,6.239,149.359
C00524=1133.120,-36.414,-47.839,179.216,6.239,149.360
C00525=1133.124,-36.664,-47.828,179.214,6.238,149.360
C00526=1133.130,-36.914,-47.816,179.211,6.237,149.360
C00527=1133.135,-37.164,-47.804,179.209,6.237,149.361
C00528=1133.141,-37.413,-47.793,179.207,6.236,149.362
C00529=1133.146,-37.663,-47.781,179.204,6.235,149.362
C00530=1133.151,-37.912,-47.770,179.202,6.235,149.363
C00531=1133.156,-38.162,-47.758,179.200,6.234,149.363
C00532=1133.161,-38.411,-47.747,179.197,6.233,149.364
C00533=1133.167,-38.662,-47.736,179.195,6.233,149.364
C00534=1133.172,-38.911,-47.725,179.193,6.232,149.365
C00535=1133.177,-39.161,-47.713,179.190,6.232,149.365
C00536=1133.183,-39.410,-47.702,179.188,6.231,149.366
C00537=1133.188,-39.660,-47.690,179.186,6.230,149.366
C00538=1133.193,-39.910,-47.679,179.183,6.230,149.367
C00539=1133.198,-40.159,-47.669,179.181,6.229,149.368
C00540=1133.204,-40.409,-47.657,179.179,6.228,149.368
C00541=1133.208,-40.659,-47.645,179.177,6.228,149.369
C00542=1133.214,-40.909,-47.634,179.175,6.228,149.369
C00543=1133.219,-41.158,-47.623,179.172,6.227,149.370
C00544=1133.225,-41.408,-47.611,179.170,6.226,149.370
C00545=1133.230,-41.658,-47.600,179.168,6.225,149.371
C00546=1133.236,-41.907,-47.589,179.165,6.225,149.371
C00547=1133.240,-42.157,-47.577,179.163,6.224,149.372
C00548=1133.245,-42.407,-47.567,179.161,6.223,149.372
C00549=1133.251,-42.657,-47.555,179.158,6.223,149.373
C00550=1133.256,-42.906,-47.544,179.156,6.222,149.373
C00551=1133.261,-43.156,-47.532,179.154,6.221,149.374
C00552=1133.266,-43.406,-47.522,179.152,6.221,149.374
C00553=1133.272,-43.655,-47.511,179.149,6.220,149.375
C00554=1133.277,-43.905,-47.499,179.147,6.220,149.376
C00555=1133.282,-44.154,-47.487,179.145,6.219,149.376
C00556=1133.287,-44.404,-47.477,179.143,6.218,149.377
C00557=1133.293,-44.654,-47.465,179.140,6.218,149.377
C00558=1133.298,-44.904,-47.454,179.138,6.217,149.378
C00559=1133.303,-45.153,-47.444,179.136,6.216,149.378
C00560=1133.309,-45.403,-47.432,179.133,6.216,149.379
C00561=1133.313,-45.653,-47.421,179.131,6.215,149.379
C00562=1133.319,-45.902,-47.410,179.128,6.214,149.380
C00563=1133.324,-46.152,-47.399,179.126,6.213,149.380
C00564=1133.330,-46.402,-47.388,179.124,6.213,149.381
C00565=1133.335,-46.651,-47.377,179.121,6.212,149.382
C00566=1133.340,-46.901,-47.365,179.119,6.211,149.382
C00567=1133.346,-47.151,-47.355,179.118,6.211,149.382
C00568=1133.350,-47.400,-47.344,179.115,6.211,149.383
C00569=1133.356,-47.651,-47.333,179.113,6.210,149.384
C00570=1133.361,-47.900,-47.322,179.111,6.209,149.384
C00571=1133.366,-48.149,-47.310,179.108,6.209,149.385
C00572=1133.372,-48.399,-47.300,179.106,6.208,149.385
C00573=1133.377,-48.649,-47.288,179.104,6.208,149.386
C00574=1133.382,-48.899,-47.278,179.101,6.207,149.386
C00575=1133.387,-49.148,-47.267,179.099,6.206,149.387
C00576=1133.393,-49.399,-47.256,179.096,6.206,149.387
C00577=1133.398,-49.648,-47.245,179.094,6.205,149.388
C00578=1133.403,-49.898,-47.234,179.092,6.204,149.388
C00579=1133.408,-50.147,-47.223,179.089,6.204,149.389
C00580=1133.414,-50.397,-47.213,179.087,6.203,149.390
C00581=1133.419,-50.668,-47.200,179.085,6.202,149.390
C00582=1133.425,-50.938,-47.188,179.082,6.202,149.391
C00583=1133.431,-51.209,-47.176,179.080,6.201,149.391
C00584=1133.436,-51.480,-47.165,179.078,6.201,149.392
C00585=1133.442,-51.730,-47.154,179.075,6.200,149.392
C00586=1133.447,-51.980,-47.143,179.073,6.199,149.393
C00587=1133.453,-52.229,-47.132,179.071,6.198,149.393
C00588=1133.458,-52.479,-47.122,179.068,6.198,149.394
C00589=1133.463,-52.728,-47.111,179.067,6.198,149.395
C00590=1133.469,-52.979,-47.100,179.065,6.197,149.395
C00591=1133.474,-53.228,-47.089,179.062,6.196,149.396
C00592=1133.479,-53.478,-47.078,179.060,6.196,149.396
C00593=1133.484,-53.728,-47.067,179.057,6.195,149.397
C00594=1133.489,-53.977,-47.057,179.055,6.194,149.397
C00595=1133.494,-54.227,-47.046,179.053,6.194,149.398
C00596=1133.500,-54.477,-47.034,179.050,6.193,149.398
C00597=1133.505,-54.727,-47.024,179.048,6.193,149.399
C00598=1133.511,-54.976,-47.014,179.046,6.192,149.399
C00599=1133.515,-55.226,-47.002,179.044,6.192,149.400
C00600=1133.521,-55.475,-46.992,179.042,6.191,149.400
C00601=1133.526,-55.726,-46.982,179.040,6.191,149.401
C00602=1133.531,-55.975,-46.971,179.037,6.190,149.402
C00603=1133.536,-56.225,-46.960,179.035,6.189,149.402
C00604=1133.542,-56.474,-46.950,179.033,6.188,149.402
C00605=1133.547,-56.724,-46.939,179.030,6.188,149.403
C00606=1133.553,-56.974,-46.928,179.028,6.187,149.404
C00607=1133.558,-57.224,-46.917,179.026,6.186,149.404
C00608=1133.563,-57.473,-46.906,179.024,6.186,149.405
C00609=1133.568,-57.723,-46.896,179.022,6.186,149.405
C00610=1133.574,-57.973,-46.886,179.020,6.185,149.406
C00611=1133.579,-58.222,-46.874,179.017,6.185,149.406
C00612=1133.584,-58.472,-46.864,179.015,6.184,149.407
C00613=1133.590,-58.722,-46.854,179.012,6.183,149.407
C00614=1133.595,-58.972,-46.843,179.010,6.183,149.408
C00615=1133.600,-59.221,-46.832,179.009,6.183,149.408
C00616=1133.605,-59.471,-46.822,179.006,6.182,149.409
C00617=1133.611,-59.721,-46.812,179.004,6.182,149.410
C00618=1133.616,-59.971,-46.801,179.002,6.181,149.410
C00619=1133.621,-60.220,-46.791,178.999,6.180,149.411
C00620=1133.626,-60.470,-46.779,178.997,6.179,149.411
C00621=1133.632,-60.719,-46.769,178.995,6.178,149.412
C00622=1133.637,-60.969,-46.759,178.992,6.178,149.412
C00623=1133.642,-61.219,-46.748,178.991,6.178,149.413
C00624=1133.648,-61.469,-46.738,178.989,6.177,149.413
C00625=1133.652,-61.718,-46.727,178.986,6.177,149.414
C00626=1133.658,-61.968,-46.717,178.984,6.176,149.414
C00627=1133.664,-62.218,-46.707,178.982,6.175,149.415
C00628=1133.669,-62.468,-46.696,178.979,6.175,149.415
C00629=1133.674,-62.717,-46.686,178.977,6.174,149.416
C00630=1133.679,-62.968,-46.675,178.976,6.174,149.416
C00631=1133.685,-63.217,-46.665,178.973,6.174,149.417
C00632=1133.690,-63.466,-46.654,178.971,6.173,149.418
C00633=1133.695,-63.716,-46.643,178.969,6.172,149.418
C00634=1133.701,-63.966,-46.633,178.966,6.171,149.418
C00635=1133.706,-64.216,-46.623,178.964,6.171,149.419
C00636=1133.711,-64.465,-46.613,178.962,6.171,149.420
C00637=1133.716,-64.715,-46.603,178.960,6.170,149.420
C00638=1133.721,-64.965,-46.592,178.958,6.169,149.421
C00639=1133.727,-65.215,-46.582,178.955,6.169,149.421
C00640=1133.732,-65.464,-46.572,178.953,6.168,149.422
C00641=1133.737,-65.714,-46.561,178.951,6.167,149.422
C00642=1133.743,-65.964,-46.551,178.949,6.167,149.423
C00643=1133.748,-66.214,-46.541,178.947,6.167,149.423
C00644=1133.754,-66.464,-46.530,178.945,6.166,149.424
C00645=1133.759,-66.713,-46.520,178.942,6.166,149.424
C00646=1133.763,-66.963,-46.510,178.940,6.165,149.425
C00647=1133.769,-67.213,-46.500,178.938,6.164,149.425
C00648=1133.775,-67.462,-46.490,178.936,6.164,149.426
C00649=1133.780,-67.713,-46.479,178.934,6.163,149.426
C00650=1133.785,-67.962,-46.469,178.931,6.163,149.427
C00651=1133.791,-68.212,-46.459,178.929,6.162,149.428
C00652=1133.796,-68.461,-46.449,178.927,6.161,149.428
C00653=1133.801,-68.711,-46.439,178.925,6.161,149.429
C00654=1133.806,-68.961,-46.428,178.923,6.161,149.429
C00655=1133.812,-69.210,-46.418,178.920,6.160,149.430
C00656=1133.817,-69.460,-46.408,178.918,6.160,149.430
C00657=1133.822,-69.710,-46.397,178.916,6.159,149.431
C00658=1133.828,-69.960,-46.387,178.914,6.158,149.431
C00659=1133.832,-70.209,-46.377,178.912,6.158,149.432
C00660=1133.838,-70.459,-46.367,178.909,6.158,149.432
C00661=1133.844,-70.709,-46.357,178.907,6.157,149.433
C00662=1133.849,-70.958,-46.347,178.905,6.156,149.433
C00663=1133.854,-71.208,-46.336,178.903,6.155,149.434
C00664=1133.859,-71.458,-46.327,178.901,6.155,149.434
C00665=1133.865,-71.708,-46.317,178.899,6.155,149.435
C00666=1133.870,-71.957,-46.307,178.896,6.154,149.435
C00667=1133.875,-72.208,-46.296,178.894,6.154,149.436
C00668=1133.881,-72.457,-46.286,178.893,6.154,149.436
C00669=1133.886,-72.706,-46.276,178.890,6.153,149.437
C00670=1133.892,-72.956,-46.266,178.888,6.152,149.438
C00671=1133.897,-73.207,-46.256,178.886,6.152,149.438
C00672=1133.902,-73.456,-46.246,178.883,6.151,149.439
C00673=1133.907,-73.705,-46.236,178.882,6.151,149.439
C00674=1133.913,-73.955,-46.226,178.880,6.150,149.440
C00675=1133.918,-74.205,-46.216,178.877,6.149,149.440
C00676=1133.924,-74.455,-46.206,178.875,6.149,149.441
C00677=1133.929,-74.705,-46.196,178.873,6.148,149.441
C00678=1133.934,-74.954,-46.186,178.871,6.148,149.442
C00679=1133.939,-75.204,-46.176,178.869,6.148,149.442
C00680=1133.944,-75.454,-46.166,178.867,6.147,149.443
C00681=1133.950,-75.704,-46.157,178.864,6.146,149.443
C00682=1133.956,-75.953,-46.146,178.862,6.146,149.444
C00683=1133.961,-76.203,-46.136,178.860,6.146,149.444
C00684=1133.965,-76.453,-46.126,178.858,6.145,149.445
C00685=1133.972,-76.724,-46.116,178.856,6.144,149.445
C00686=1133.977,-76.996,-46.105,178.853,6.144,149.446
C00687=1133.983,-77.268,-46.095,178.851,6.143,149.447
C00688=1133.990,-77.539,-46.083,178.849,6.142,149.447
C00689=1133.995,-77.789,-46.074,178.847,6.143,149.448
C00690=1134.000,-78.039,-46.064,178.844,6.142,149.448
C00691=1134.005,-78.288,-46.054,178.842,6.141,149.449
C00692=1134.010,-78.538,-46.045,178.840,6.140,149.449
C00693=1134.016,-78.788,-46.035,178.838,6.141,149.450
C00694=1134.022,-79.037,-46.024,178.836,6.140,149.450
C00695=1134.026,-79.288,-46.015,178.834,6.139,149.451
C00696=1134.032,-79.537,-46.005,178.831,6.139,149.451
C00697=1134.037,-79.787,-45.995,178.829,6.138,149.452
C00698=1134.043,-80.037,-45.986,178.828,6.138,149.452
C00699=1134.048,-80.286,-45.976,178.825,6.137,149.453
C00700=1134.053,-80.535,-45.966,178.823,6.136,149.453
C00701=1134.059,-80.786,-45.956,178.821,6.137,149.454
C00702=1134.064,-81.036,-45.946,178.819,6.136,149.454
C00703=1134.069,-81.285,-45.936,178.817,6.135,149.455
C00704=1134.075,-81.535,-45.927,178.814,6.135,149.455
C00705=1134.080,-81.784,-45.917,178.813,6.135,149.456
C00706=1134.085,-82.035,-45.908,178.811,6.134,149.456
C00707=1134.091,-82.284,-45.897,178.808,6.133,149.457
C00708=1134.096,-82.534,-45.889,178.806,6.133,149.458
C00709=1134.102,-82.783,-45.878,178.804,6.133,149.458
C00710=1134.106,-83.033,-45.868,178.802,6.132,149.459
C00711=1134.112,-83.284,-45.859,178.800,6.131,149.459
C00712=1134.117,-83.533,-45.849,178.798,6.130,149.460
C00713=1134.123,-83.783,-45.840,178.796,6.131,149.460
C00714=1134.128,-84.032,-45.830,178.793,6.130,149.461
C00715=1134.134,-84.282,-45.821,178.791,6.129,149.461
C00716=1134.138,-84.532,-45.811,178.789,6.129,149.462
C00717=1134.144,-84.782,-45.802,178.787,6.129,149.462
C00718=1134.149,-85.031,-45.792,178.785,6.128,149.463
C00719=1134.155,-85.281,-45.782,178.783,6.127,149.463
C00720=1134.159,-85.531,-45.773,178.781,6.127,149.464
C00721=1134.165,-85.781,-45.763,178.779,6.127,149.464
C00722=1134.170,-86.030,-45.753,178.777,6.126,149.465
C00723=1134.176,-86.281,-45.744,178.774,6.125,149.465
C00724=1134.181,-86.530,-45.734,178.773,6.125,149.466
C00725=1134.187,-86.780,-45.725,178.771,6.125,149.466
C00726=1134.192,-87.029,-45.715,178.768,6.124,149.467
C00727=1134.197,-87.279,-45.706,178.767,6.124,149.467
C00728=1134.203,-87.529,-45.697,178.765,6.123,149.468
C00729=1134.208,-87.779,-45.687,178.762,6.123,149.468
C00730=1134.213,-88.029,-45.678,178.760,6.122,149.469
C00731=1134.218,-88.278,-45.668,178.758,6.122,149.469
C00732=1134.224,-88.528,-45.659,178.756,6.121,149.470
C00733=1134.229,-88.777,-45.649,178.754,6.121,149.470
C00734=1134.235,-89.027,-45.639,178.752,6.121,149.471
C00735=1134.240,-89.277,-45.631,178.750,6.120,149.471
C00736=1134.246,-89.527,-45.620,178.748,6.119,149.472
C00737=1134.251,-89.777,-45.611,178.746,6.120,149.473
C00738=1134.256,-90.027,-45.603,178.743,6.119,149.473
C00739=1134.262,-90.276,-45.592,178.741,6.118,149.473
C00740=1134.266,-90.527,-45.583,178.739,6.117,149.474
C00741=1134.272,-90.776,-45.573,178.737,6.117,149.474
C00742=1134.277,-91.026,-45.564,178.735,6.117,149.475
C00743=1134.282,-91.276,-45.555,178.733,6.116,149.475
C00744=1134.288,-91.525,-45.545,178.732,6.116,149.476
C00745=1134.293,-91.775,-45.536,178.729,6.115,149.476
C00746=1134.298,-92.025,-45.527,178.727,6.115,149.477
C00747=1134.304,-92.275,-45.518,178.725,6.115,149.478
C00748=1134.309,-92.524,-45.508,178.723,6.114,149.478
C00749=1134.315,-92.774,-45.499,178.721,6.113,149.479
C00750=1134.321,-93.024,-45.490,178.719,6.113,149.479
C00751=1134.325,-93.273,-45.480,178.717,6.113,149.480
C00752=1134.331,-93.523,-45.471,178.715,6.112,149.480
C00753=1134.336,-93.773,-45.462,178.713,6.112,149.480
C00754=1134.342,-94.023,-45.453,178.711,6.111,149.481
C00755=1134.347,-94.273,-45.443,178.708,6.111,149.482
C00756=1134.352,-94.522,-45.434,178.706,6.110,149.482
C00757=1134.358,-94.772,-45.425,178.704,6.110,149.483
C00758=1134.363,-95.022,-45.416,178.702,6.109,149.483
C00759=1134.368,-95.272,-45.406,178.700,6.108,149.484
C00760=1134.373,-95.521,-45.397,178.698,6.109,149.484
C00761=1134.379,-95.771,-45.388,178.696,6.108,149.485
C00762=1134.385,-96.021,-45.379,178.694,6.107,149.485
C00763=1134.390,-96.271,-45.370,178.692,6.107,149.486
C00764=1134.395,-96.521,-45.360,178.690,6.106,149.486
C00765=1134.400,-96.771,-45.351,178.688,6.106,149.487
C00766=1134.406,-97.021,-45.342,178.686,6.106,149.487
C00767=1134.411,-97.270,-45.333,178.684,6.105,149.488
C00768=1134.417,-97.520,-45.324,178.682,6.105,149.488
C00769=1134.422,-97.770,-45.315,178.680,6.105,149.489
C00770=1134.427,-98.019,-45.305,178.678,6.104,149.489
C00771=1134.433,-98.269,-45.296,178.676,6.104,149.490
C00772=1134.438,-98.519,-45.287,178.674,6.103,149.490
C00773=1134.444,-98.769,-45.278,178.672,6.102,149.491
C00774=1134.449,-99.019,-45.269,178.670,6.102,149.491
C00775=1134.454,-99.269,-45.260,178.668,6.102,149.492
C00776=1134.459,-99.518,-45.251,178.666,6.101,149.492
C00777=1134.465,-99.768,-45.241,178.664,6.101,149.493
C00778=1134.470,-100.017,-45.232,178.662,6.100,149.493
C00779=1134.476,-100.267,-45.224,178.659,6.100,149.494
C00780=1134.481,-100.517,-45.215,178.658,6.100,149.494
C00781=1134.487,-100.767,-45.205,178.656,6.099,149.495
C00782=1134.492,-101.017,-45.196,178.653,6.098,149.495
C00783=1134.497,-101.267,-45.187,178.652,6.098,149.496
C00784=1134.502,-101.516,-45.179,178.650,6.098,149.496
C00785=1134.507,-101.766,-45.170,178.648,6.098,149.497
C00786=1134.513,-102.015,-45.161,178.646,6.097,149.497
C00787=1134.519,-102.266,-45.152,178.644,6.096,149.498
C00788=1134.524,-102.516,-45.143,178.642,6.096,149.498
C00789=1134.530,-102.787,-45.132,178.640,6.095,149.499
C00790=1134.535,-103.060,-45.123,178.637,6.095,149.499
C00791=1134.541,-103.333,-45.113,178.635,6.094,149.500
C00792=1134.547,-103.604,-45.103,178.633,6.094,149.500
C00793=1134.553,-103.854,-45.095,178.631,6.094,149.501
C00794=1134.558,-104.103,-45.086,178.629,6.093,149.501
C00795=1134.564,-104.354,-45.076,178.627,6.093,149.502
C00796=1134.569,-104.603,-45.067,178.625,6.092,149.502
C00797=1134.574,-104.853,-45.059,178.623,6.091,149.503
C00798=1134.579,-105.103,-45.050,178.621,6.092,149.503
C00799=1134.585,-105.352,-45.041,178.619,6.091,149.504
C00800=1134.590,-105.603,-45.033,178.618,6.091,149.504
C00801=1134.596,-105.853,-45.024,178.615,6.090,149.505
C00802=1134.601,-106.103,-45.015,178.613,6.090,149.505
C00803=1134.606,-106.352,-45.006,178.611,6.090,149.506
C00804=1134.611,-106.602,-44.997,178.609,6.089,149.506
C00805=1134.618,-106.852,-44.988,178.607,6.088,149.507
C00806=1134.623,-107.102,-44.979,178.605,6.088,149.507
C00807=1134.628,-107.351,-44.970,178.603,6.088,149.508
C00808=1134.633,-107.601,-44.961,178.601,6.088,149.508
C00809=1134.639,-107.850,-44.953,178.599,6.087,149.509
C00810=1134.644,-108.100,-44.944,178.597,6.086,149.509
C00811=1134.649,-108.350,-44.935,178.595,6.086,149.510
C00812=1134.655,-108.601,-44.927,178.593,6.085,149.510
C00813=1134.660,-108.850,-44.918,178.591,6.085,149.511
C00814=1134.666,-109.100,-44.910,178.589,6.085,149.511
C00815=1134.671,-109.349,-44.901,178.587,6.084,149.512
C00816=1134.676,-109.599,-44.892,178.586,6.084,149.512
C00817=1134.681,-109.849,-44.883,178.583,6.083,149.513
C00818=1134.687,-110.098,-44.874,178.582,6.083,149.513
C00819=1134.692,-110.349,-44.866,178.580,6.083,149.514
C00820=1134.697,-110.599,-44.857,178.577,6.082,149.514
C00821=1134.703,-110.848,-44.848,178.576,6.082,149.515
C00822=1134.708,-111.098,-44.840,178.574,6.081,149.515
C00823=1134.714,-111.347,-44.831,178.572,6.081,149.516
C00824=1134.719,-111.598,-44.823,178.570,6.080,149.516
C00825=1134.724,-111.848,-44.814,178.568,6.080,149.517
C00826=1134.730,-112.097,-44.805,178.566,6.080,149.517
C00827=1134.735,-112.347,-44.796,178.564,6.079,149.518
C00828=1134.740,-112.597,-44.787,178.562,6.079,149.518
C00829=1134.746,-112.847,-44.779,178.560,6.078,149.519
C00830=1134.752,-113.096,-44.771,178.558,6.078,149.519
C00831=1134.757,-113.346,-44.762,178.556,6.078,149.520
C00832=1134.762,-113.596,-44.753,178.554,6.077,149.520
C00833=1134.768,-113.846,-44.745,178.552,6.077,149.521
C00834=1134.773,-114.096,-44.736,178.550,6.076,149.521
C00835=1134.778,-114.345,-44.727,178.549,6.076,149.522
C00836=1134.783,-114.595,-44.718,178.546,6.075,149.522
C00837=1134.789,-114.845,-44.711,178.545,6.075,149.522
C00838=1134.795,-115.095,-44.702,178.543,6.075,149.523
C00839=1134.800,-115.345,-44.693,178.540,6.074,149.523
C00840=1134.806,-115.594,-44.685,178.539,6.074,149.524
C00841=1134.811,-115.844,-44.676,178.537,6.073,149.524
C00842=1134.816,-116.094,-44.667,178.535,6.073,149.525
C00843=1134.822,-116.344,-44.659,178.533,6.073,149.525
C00844=1134.827,-116.593,-44.651,178.531,6.073,149.526
C00845=1134.832,-116.843,-44.642,178.529,6.072,149.526
C00846=1134.838,-117.093,-44.634,178.527,6.072,149.527
C00847=1134.843,-117.343,-44.626,178.525,6.071,149.527
C00848=1134.848,-117.593,-44.617,178.523,6.070,149.528
C00849=1134.854,-117.843,-44.609,178.521,6.070,149.528
C00850=1134.860,-118.092,-44.600,178.519,6.070,149.529
C00851=1134.865,-118.342,-44.591,178.518,6.070,149.529
C00852=1134.871,-118.592,-44.583,178.515,6.069,149.530
C00853=1134.875,-118.842,-44.575,178.514,6.069,149.530
C00854=1134.880,-119.091,-44.566,178.512,6.068,149.531
C00855=1134.886,-119.341,-44.558,178.510,6.068,149.531
C00856=1134.892,-119.591,-44.549,178.508,6.068,149.532
C00857=1134.898,-119.841,-44.541,178.506,6.067,149.532
C00858=1134.903,-120.091,-44.533,178.504,6.067,149.533
C00859=1134.908,-120.341,-44.524,178.502,6.066,149.533
C00860=1134.913,-120.590,-44.516,178.500,6.066,149.534
C00861=1134.919,-120.840,-44.508,178.498,6.066,149.534
C00862=1134.924,-121.090,-44.499,178.496,6.066,149.535
C00863=1134.930,-121.339,-44.491,178.494,6.065,149.535
C00864=1134.935,-121.590,-44.483,178.493,6.065,149.536
C00865=1134.940,-121.839,-44.474,178.490,6.064,149.536
C00866=1134.946,-122.089,-44.467,178.489,6.064,149.536
C00867=1134.951,-122.339,-44.458,178.487,6.063,149.537
C00868=1134.957,-122.588,-44.449,178.485,6.062,149.537
C00869=1134.962,-122.839,-44.441,178.483,6.062,149.538
C00870=1134.967,-123.088,-44.433,178.481,6.062,149.538
C00871=1134.973,-123.338,-44.425,178.480,6.062,149.539
C00872=1134.978,-123.588,-44.416,178.477,6.061,149.539
C00873=1134.984,-123.838,-44.408,178.476,6.061,149.540
C00874=1134.989,-124.087,-44.399,178.474,6.060,149.540
C00875=1134.994,-124.337,-44.392,178.472,6.060,149.541
C00876=1135.000,-124.587,-44.383,178.470,6.060,149.541
C00877=1135.005,-124.837,-44.375,178.468,6.060,149.542
C00878=1135.011,-125.087,-44.367,178.466,6.059,149.542
C00879=1135.016,-125.337,-44.359,178.464,6.059,149.543
C00880=1135.022,-125.586,-44.351,178.462,6.058,149.543
C00881=1135.027,-125.836,-44.342,178.461,6.058,149.544
C00882=1135.033,-126.086,-44.334,178.458,6.057,149.544
C00883=1135.037,-126.336,-44.326,178.457,6.057,149.544
C00884=1135.043,-126.586,-44.318,178.455,6.056,149.545
C00885=1135.049,-126.835,-44.309,178.453,6.056,149.545
C00886=1135.054,-127.086,-44.301,178.451,6.056,149.546
C00887=1135.059,-127.335,-44.294,178.450,6.056,149.546
C00888=1135.064,-127.585,-44.285,178.447,6.055,149.547
C00889=1135.071,-127.835,-44.277,178.446,6.055,149.547
C00890=1135.075,-128.084,-44.269,178.444,6.054,149.548
C00891=1135.081,-128.334,-44.261,178.441,6.054,149.548
C00892=1135.087,-128.584,-44.253,178.440,6.054,149.549
C00893=1134.665,-128.596,-44.297,178.437,6.057,149.550
C00894=1134.660,-128.345,-44.305,178.439,6.057,149.550
C00895=1134.655,-128.096,-44.312,178.440,6.058,149.550
C00896=1134.649,-127.846,-44.321,178.442,6.058,149.549
C00897=1134.643,-127.596,-44.329,178.444,6.059,149.549
C00898=1134.638,-127.346,-44.338,178.446,6.059,149.548
C00899=1134.633,-127.097,-44.345,178.448,6.060,149.548
C00900=1134.627,-126.846,-44.353,178.450,6.060,149.547
C00901=1134.622,-126.597,-44.362,178.452,6.060,149.547
C00902=1134.617,-126.347,-44.369,178.453,6.060,149.546
C00903=1134.611,-126.098,-44.378,178.456,6.061,149.546
C00904=1134.606,-125.847,-44.386,178.457,6.061,149.545
C00905=1134.601,-125.597,-44.395,178.459,6.062,149.545
C00906=1134.595,-125.348,-44.402,178.461,6.062,149.544
C00907=1134.590,-125.098,-44.411,178.463,6.063,149.544
C00908=1134.584,-124.848,-44.419,178.464,6.063,149.544
C00909=1134.578,-124.598,-44.427,178.467,6.064,149.543
C00910=1134.573,-124.349,-44.435,178.468,6.064,149.543
C00911=1134.568,-124.099,-44.443,178.470,6.064,149.542
C00912=1134.563,-123.849,-44.452,178.472,6.064,149.542
C00913=1134.557,-123.599,-44.460,178.474,6.065,149.541
C00914=1134.552,-123.349,-44.468,178.476,6.065,149.541
C00915=1134.546,-123.100,-44.476,178.478,6.066,149.540
C00916=1134.541,-122.850,-44.485,178.479,6.066,149.540
C00917=1134.536,-122.599,-44.493,178.482,6.066,149.539
C00918=1134.530,-122.350,-44.502,178.484,6.067,149.539
C00919=1134.525,-122.100,-44.509,178.485,6.067,149.538
C00920=1134.519,-121.851,-44.518,178.488,6.068,149.538
C00921=1134.514,-121.601,-44.527,178.489,6.068,149.537
C00922=1134.509,-121.351,-44.535,178.491,6.069,149.537
C00923=1134.503,-121.101,-44.543,178.493,6.068,149.536
C00924=1134.498,-120.851,-44.551,178.495,6.069,149.536
C00925=1134.493,-120.601,-44.560,178.497,6.069,149.535
C00926=1134.487,-120.352,-44.568,178.499,6.070,149.535
C00927=1134.482,-120.102,-44.577,178.500,6.070,149.535
C00928=1134.476,-119.853,-44.585,178.502,6.071,149.534
C00929=1134.471,-119.602,-44.593,178.505,6.072,149.534
C00930=1134.466,-119.353,-44.602,178.506,6.072,149.533
C00931=1134.460,-119.103,-44.610,178.508,6.072,149.533
C00932=1134.455,-118.853,-44.618,178.510,6.072,149.532
C00933=1134.450,-118.603,-44.627,178.512,6.073,149.532
C00934=1134.444,-118.353,-44.635,178.514,6.073,149.531
C00935=1134.438,-118.104,-44.644,178.516,6.074,149.531
C00936=1134.433,-117.853,-44.652,178.518,6.074,149.530
C00937=1134.427,-117.604,-44.661,178.520,6.075,149.530
C00938=1134.423,-117.354,-44.669,178.522,6.075,149.529
C00939=1134.417,-117.104,-44.677,178.524,6.075,149.529
C00940=1134.412,-116.855,-44.686,178.526,6.076,149.528
C00941=1134.406,-116.605,-44.695,178.527,6.076,149.528
C00942=1134.401,-116.354,-44.703,178.530,6.077,149.527
C00943=1134.395,-116.105,-44.711,178.531,6.077,149.527
C00944=1134.390,-115.855,-44.720,178.533,6.077,149.526
C00945=1134.385,-115.605,-44.728,178.535,6.077,149.526
C00946=1134.379,-115.356,-44.737,178.537,6.078,149.525
C00947=1134.374,-115.106,-44.746,178.539,6.079,149.525
C00948=1134.368,-114.856,-44.755,178.541,6.079,149.524
C00949=1134.362,-114.606,-44.763,178.543,6.079,149.524
C00950=1134.357,-114.356,-44.772,178.545,6.079,149.523
C00951=1134.353,-114.107,-44.780,178.547,6.080,149.523
C00952=1134.347,-113.857,-44.788,178.549,6.080,149.522
C00953=1134.342,-113.607,-44.797,178.551,6.081,149.522
C00954=1134.336,-113.357,-44.805,178.553,6.082,149.521
C00955=1134.331,-113.108,-44.814,178.555,6.082,149.521
C00956=1134.325,-112.858,-44.822,178.557,6.082,149.520
C00957=1134.320,-112.608,-44.831,178.558,6.082,149.520
C00958=1134.315,-112.358,-44.840,178.561,6.083,149.519
C00959=1134.309,-112.109,-44.848,178.563,6.084,149.519
C00960=1134.304,-111.859,-44.857,178.564,6.084,149.518
C00961=1134.298,-111.609,-44.866,178.567,6.084,149.518
C00962=1134.293,-111.359,-44.874,178.568,6.084,149.517
C00963=1134.287,-111.110,-44.883,178.570,6.085,149.517
C00964=1134.282,-110.860,-44.892,178.572,6.085,149.517
C00965=1134.277,-110.610,-44.901,178.574,6.086,149.516
C00966=1134.272,-110.360,-44.909,178.576,6.087,149.516
C00967=1134.266,-110.110,-44.917,178.578,6.087,149.515
C00968=1134.261,-109.861,-44.926,178.580,6.087,149.515
C00969=1134.256,-109.611,-44.935,178.582,6.087,149.514
C00970=1134.250,-109.361,-44.944,178.584,6.088,149.514
C00971=1134.245,-109.112,-44.953,178.586,6.089,149.513
C00972=1134.239,-108.861,-44.961,178.588,6.089,149.513
C00973=1134.233,-108.611,-44.970,178.590,6.089,149.512
C00974=1134.228,-108.361,-44.979,178.591,6.089,149.512
C00975=1134.223,-108.111,-44.988,178.594,6.090,149.511
C00976=1134.217,-107.862,-44.997,178.596,6.091,149.511
C00977=1134.212,-107.612,-45.006,178.597,6.091,149.510
C00978=1134.207,-107.362,-45.015,178.600,6.092,149.510
C00979=1134.202,-107.113,-45.023,178.601,6.092,149.509
C00980=1134.196,-106.863,-45.032,178.603,6.092,149.509
C00981=1134.190,-106.613,-45.040,178.606,6.093,149.508
C00982=1134.185,-106.363,-45.049,178.607,6.093,149.508
C00983=1134.180,-106.113,-45.058,178.609,6.094,149.507
C00984=1134.175,-105.863,-45.067,178.612,6.095,149.507
C00985=1134.170,-105.614,-45.076,178.613,6.094,149.506
C00986=1134.163,-105.364,-45.085,178.616,6.095,149.506
C00987=1134.158,-105.114,-45.094,178.617,6.095,149.505
C00988=1134.153,-104.864,-45.103,178.620,6.096,149.505
C00989=1134.148,-104.615,-45.112,178.622,6.096,149.504
C00990=1134.143,-104.365,-45.120,178.623,6.096,149.504
C00991=1134.137,-104.116,-45.129,178.626,6.097,149.503
C00992=1134.132,-103.866,-45.138,178.627,6.097,149.503
C00993=1134.126,-103.616,-45.147,178.629,6.098,149.502
C00994=1134.121,-103.343,-45.156,178.632,6.098,149.502
C00995=1134.114,-103.071,-45.167,178.634,6.099,149.501
C00996=1134.109,-102.799,-45.177,178.636,6.099,149.500
C00997=1134.103,-102.526,-45.186,178.638,6.099,149.500
C00998=1134.097,-102.277,-45.195,178.640,6.100,149.499
C00999=1134.092,-102.027,-45.204,178.642,6.100,149.499
C01000=1134.087,-101.777,-45.212,178.644,6.101,149.499
C01001=1134.082,-101.528,-45.222,178.646,6.102,149.498
C01002=1134.076,-101.278,-45.232,178.648,6.102,149.498
C01003=1134.071,-101.028,-45.240,178.650,6.102,149.497
C01004=1134.066,-100.778,-45.249,178.652,6.103,149.497
C01005=1134.060,-100.528,-45.258,178.654,6.103,149.496
C01006=1134.055,-100.279,-45.267,178.656,6.104,149.496
C01007=1134.049,-100.029,-45.276,178.658,6.105,149.495
C01008=1134.044,-99.779,-45.285,178.660,6.105,149.495
C01009=1134.038,-99.529,-45.294,178.663,6.105,149.494
C01010=1134.033,-99.279,-45.303,178.665,6.106,149.493
C01011=1134.028,-99.029,-45.312,178.666,6.106,149.493
C01012=1134.023,-98.780,-45.322,178.669,6.106,149.492
C01013=1134.017,-98.530,-45.331,178.671,6.107,149.492
C01014=1134.012,-98.280,-45.340,178.672,6.107,149.492
C01015=1134.006,-98.031,-45.348,178.675,6.108,149.491
C01016=1134.001,-97.781,-45.358,178.676,6.108,149.491
C01017=1133.995,-97.531,-45.367,178.678,6.109,149.490
C01018=1133.990,-97.281,-45.376,178.681,6.109,149.490
C01019=1133.985,-97.032,-45.386,178.682,6.109,149.489
C01020=1133.979,-96.782,-45.395,178.684,6.110,149.489
C01021=1133.974,-96.532,-45.404,178.687,6.111,149.488
C01022=1133.969,-96.282,-45.413,178.689,6.110,149.487
C01023=1133.963,-96.032,-45.422,178.691,6.111,149.487
C01024=1133.958,-95.782,-45.431,178.693,6.112,149.486
C01025=1133.953,-95.533,-45.441,178.695,6.112,149.486
C01026=1133.947,-95.283,-45.450,178.697,6.113,149.485
C01027=1133.942,-95.033,-45.459,178.699,6.113,149.485
C01028=1133.936,-94.784,-45.468,178.701,6.113,149.484
C01029=1133.931,-94.534,-45.477,178.703,6.114,149.484
C01030=1133.926,-94.284,-45.487,178.705,6.115,149.484
C01031=1133.920,-94.034,-45.496,178.707,6.115,149.483
C01032=1133.915,-93.785,-45.504,178.709,6.115,149.483
C01033=1133.910,-93.535,-45.515,178.711,6.116,149.482
C01034=1133.904,-93.285,-45.524,178.713,6.116,149.481
C01035=1133.899,-93.035,-45.532,178.715,6.117,149.481
C01036=1133.893,-92.785,-45.542,178.717,6.117,149.480
C01037=1133.889,-92.536,-45.552,178.720,6.118,149.480
C01038=1133.883,-92.286,-45.561,178.721,6.118,149.479
C01039=1133.877,-92.036,-45.570,178.723,6.119,149.479
C01040=1133.873,-91.787,-45.580,178.726,6.120,149.478
C01041=1133.867,-91.537,-45.589,178.727,6.119,149.478
C01042=1133.862,-91.287,-45.598,178.729,6.120,149.477
C01043=1133.857,-91.037,-45.608,178.732,6.121,149.477
C01044=1133.851,-90.787,-45.617,178.734,6.121,149.476
C01045=1133.846,-90.537,-45.626,178.736,6.121,149.476
C01046=1133.840,-90.288,-45.636,178.738,6.122,149.475
C01047=1133.835,-90.038,-45.645,178.740,6.122,149.475
C01048=1133.830,-89.788,-45.654,178.742,6.123,149.474
C01049=1133.824,-89.539,-45.664,178.744,6.124,149.474
C01050=1133.819,-89.289,-45.673,178.746,6.124,149.473
C01051=1133.813,-89.039,-45.683,178.748,6.124,149.473
C01052=1133.808,-88.789,-45.692,178.751,6.125,149.472
C01053=1133.803,-88.540,-45.701,178.753,6.125,149.472
C01054=1133.797,-88.290,-45.711,178.754,6.125,149.471
C01055=1133.792,-88.040,-45.720,178.756,6.126,149.471
C01056=1133.786,-87.790,-45.730,178.759,6.127,149.470
C01057=1133.782,-87.540,-45.740,178.760,6.127,149.470
C01058=1133.776,-87.290,-45.749,178.762,6.128,149.469
C01059=1133.771,-87.041,-45.759,178.765,6.128,149.469
C01060=1133.765,-86.791,-45.768,178.767,6.129,149.468
C01061=1133.760,-86.541,-45.778,178.769,6.129,149.468
C01062=1133.755,-86.291,-45.787,178.771,6.129,149.467
C01063=1133.750,-86.042,-45.797,178.773,6.130,149.467
C01064=1133.745,-85.792,-45.806,178.775,6.130,149.466
C01065=1133.739,-85.543,-45.816,178.777,6.131,149.466
C01066=1133.734,-85.293,-45.825,178.779,6.132,149.465
C01067=1133.728,-85.043,-45.835,178.782,6.132,149.465
C01068=1133.723,-84.793,-45.844,178.784,6.132,149.464
C01069=1133.717,-84.544,-45.854,178.786,6.133,149.463
C01070=1133.713,-84.293,-45.864,178.788,6.133,149.463
C01071=1133.707,-84.044,-45.874,178.790,6.134,149.463
C01072=1133.702,-83.794,-45.883,178.792,6.134,149.462
C01073=1133.697,-83.544,-45.893,178.794,6.135,149.462
C01074=1133.691,-83.294,-45.902,178.796,6.136,149.461
C01075=1133.686,-83.045,-45.912,178.798,6.135,149.460
C01076=1133.680,-82.795,-45.921,178.800,6.136,149.460
C01077=1133.675,-82.545,-45.931,178.803,6.137,149.459
C01078=1133.669,-82.295,-45.941,178.805,6.138,149.459
C01079=1133.665,-82.045,-45.951,178.806,6.137,149.458
C01080=1133.659,-81.796,-45.961,178.809,6.138,149.458
C01081=1133.654,-81.546,-45.970,178.811,6.139,149.457
C01082=1133.648,-81.296,-45.980,178.813,6.139,149.457
C01083=1133.643,-81.046,-45.989,178.815,6.139,149.456
C01084=1133.638,-80.797,-45.999,178.817,6.140,149.456
C01085=1133.632,-80.547,-46.009,178.819,6.141,149.455
C01086=1133.627,-80.298,-46.018,178.822,6.142,149.455
C01087=1133.622,-80.047,-46.029,178.823,6.142,149.454
C01088=1133.616,-79.797,-46.038,178.826,6.142,149.454
C01089=1133.611,-79.548,-46.048,178.828,6.143,149.453
C01090=1133.606,-79.298,-46.058,178.830,6.143,149.453
C01091=1133.600,-79.049,-46.067,178.832,6.143,149.452
C01092=1133.595,-78.799,-46.077,178.834,6.144,149.452
C01093=1133.590,-78.549,-46.088,178.836,6.145,149.451
C01094=1133.585,-78.299,-46.097,178.838,6.146,149.451
C01095=1133.579,-78.049,-46.107,178.841,6.145,149.450
C01096=1133.573,-77.800,-46.117,178.843,6.146,149.450
C01097=1133.569,-77.551,-46.127,178.845,6.147,149.449
C01098=1133.562,-77.278,-46.137,178.847,6.148,149.449
C01099=1133.557,-77.007,-46.148,178.850,6.148,149.448
C01100=1133.550,-76.736,-46.159,178.852,6.149,149.447
C01101=1133.545,-76.464,-46.170,178.854,6.149,149.447
C01102=1133.539,-76.214,-46.179,178.856,6.149,149.446
C01103=1133.534,-75.965,-46.189,178.858,6.150,149.446
C01104=1133.529,-75.715,-46.199,178.861,6.150,149.445
C01105=1133.524,-75.465,-46.210,178.863,6.151,149.445
C01106=1133.518,-75.215,-46.219,178.865,6.152,149.444
C01107=1133.513,-74.966,-46.229,178.867,6.152,149.444
C01108=1133.507,-74.716,-46.239,178.869,6.152,149.443
C01109=1133.502,-74.466,-46.249,178.871,6.153,149.443
C01110=1133.498,-74.217,-46.259,178.874,6.154,149.442
C01111=1133.492,-73.967,-46.269,178.875,6.154,149.442
C01112=1133.486,-73.717,-46.279,178.877,6.155,149.441
C01113=1133.481,-73.467,-46.289,178.880,6.155,149.441
C01114=1133.476,-73.218,-46.299,178.882,6.156,149.440
C01115=1133.471,-72.968,-46.309,178.885,6.156,149.439
C01116=1133.465,-72.718,-46.319,178.886,6.156,149.439
C01117=1133.460,-72.468,-46.329,178.888,6.157,149.438
C01118=1133.455,-72.218,-46.339,178.891,6.158,149.438
C01119=1133.449,-71.969,-46.349,178.893,6.158,149.437
C01120=1133.444,-71.719,-46.359,178.895,6.159,149.437
C01121=1133.439,-71.469,-46.370,178.897,6.159,149.436
C01122=1133.433,-71.219,-46.380,178.899,6.160,149.436
C01123=1133.428,-70.970,-46.389,178.901,6.161,149.435
C01124=1133.422,-70.720,-46.399,178.904,6.161,149.435
C01125=1133.417,-70.470,-46.410,178.906,6.162,149.434
C01126=1133.412,-70.220,-46.420,178.908,6.162,149.434
C01127=1133.406,-69.971,-46.430,178.910,6.162,149.433
C01128=1133.402,-69.721,-46.440,178.912,6.163,149.433
C01129=1133.396,-69.471,-46.450,178.914,6.164,149.432
C01130=1133.391,-69.222,-46.461,178.917,6.164,149.432
C01131=1133.385,-68.972,-46.471,178.919,6.164,149.431
C01132=1133.380,-68.722,-46.481,178.921,6.165,149.431
C01133=1133.374,-68.472,-46.492,178.923,6.166,149.430
C01134=1133.370,-68.223,-46.501,178.925,6.167,149.430
C01135=1133.365,-67.973,-46.512,178.928,6.167,149.429
C01136=1133.359,-67.723,-46.522,178.930,6.168,149.428
C01137=1133.353,-67.474,-46.532,178.932,6.168,149.428
C01138=1133.348,-67.224,-46.543,178.934,6.168,149.427
C01139=1133.343,-66.974,-46.553,178.936,6.169,149.427
C01140=1133.337,-66.724,-46.563,178.939,6.170,149.426
C01141=1133.333,-66.475,-46.573,178.941,6.170,149.426
C01142=1133.327,-66.225,-46.583,178.943,6.170,149.425
C01143=1133.322,-65.975,-46.594,178.945,6.171,149.425
C01144=1133.317,-65.725,-46.604,178.947,6.172,149.424
C01145=1133.311,-65.476,-46.614,178.950,6.172,149.424
C01146=1133.306,-65.226,-46.625,178.952,6.173,149.423
C01147=1133.301,-64.976,-46.635,178.954,6.174,149.423
C01148=1133.295,-64.726,-46.645,178.956,6.174,149.422
C01149=1133.289,-64.477,-46.656,178.958,6.174,149.421
C01150=1133.284,-64.227,-46.666,178.960,6.175,149.421
C01151=1133.279,-63.977,-46.676,178.963,6.176,149.421
C01152=1133.274,-63.727,-46.686,178.965,6.176,149.420
C01153=1133.269,-63.478,-46.697,178.967,6.177,149.420
C01154=1133.264,-63.229,-46.707,178.970,6.178,149.419
C01155=1133.259,-62.978,-46.718,178.971,6.178,149.418
C01156=1133.253,-62.729,-46.728,178.973,6.178,149.418
C01157=1133.248,-62.479,-46.739,178.976,6.179,149.417
C01158=1133.242,-62.229,-46.749,178.978,6.180,149.417
C01159=1133.237,-61.979,-46.759,178.981,6.180,149.416
C01160=1133.232,-61.729,-46.770,178.983,6.181,149.416
C01161=1133.227,-61.480,-46.781,178.985,6.182,149.415
C01162=1133.222,-61.230,-46.791,178.986,6.182,149.415
C01163=1133.216,-60.981,-46.801,178.989,6.182,149.414
C01164=1133.210,-60.731,-46.812,178.991,6.183,149.414
C01165=1133.205,-60.481,-46.822,178.994,6.184,149.413
C01166=1133.200,-60.231,-46.832,178.996,6.184,149.413
C01167=1133.195,-59.982,-46.844,178.998,6.185,149.412
C01168=1133.189,-59.732,-46.854,179.001,6.186,149.411
C01169=1133.184,-59.482,-46.865,179.002,6.185,149.411
C01170=1133.179,-59.232,-46.875,179.004,6.186,149.410
C01171=1133.174,-58.983,-46.886,179.007,6.187,149.410
C01172=1133.169,-58.733,-46.896,179.009,6.187,149.409
C01173=1133.163,-58.484,-46.906,179.011,6.188,149.409
C01174=1133.158,-58.233,-46.917,179.014,6.189,149.408
C01175=1133.153,-57.984,-46.928,179.016,6.190,149.408
C01176=1133.148,-57.734,-46.939,179.018,6.190,149.407
C01177=1133.142,-57.485,-46.949,179.020,6.190,149.407
C01178=1133.137,-57.234,-46.959,179.022,6.191,149.406
C01179=1133.132,-56.985,-46.970,179.024,6.192,149.406
C01180=1133.126,-56.735,-46.981,179.027,6.192,149.405
C01181=1133.120,-56.485,-46.992,179.029,6.193,149.405
C01182=1133.116,-56.236,-47.003,179.032,6.194,149.404
C01183=1133.110,-55.986,-47.013,179.034,6.194,149.404
C01184=1133.105,-55.736,-47.024,179.036,6.195,149.403
C01185=1133.100,-55.487,-47.035,179.038,6.195,149.402
C01186=1133.095,-55.237,-47.045,179.040,6.195,149.402
C01187=1133.089,-54.987,-47.055,179.042,6.196,149.401
C01188=1133.085,-54.738,-47.067,179.045,6.197,149.401
C01189=1133.079,-54.488,-47.077,179.047,6.197,149.400
C01190=1133.074,-54.238,-47.089,179.049,6.198,149.400
C01191=1133.068,-53.989,-47.099,179.052,6.199,149.399
C01192=1133.063,-53.738,-47.110,179.054,6.200,149.399
C01193=1133.058,-53.489,-47.121,179.056,6.200,149.398
C01194=1133.053,-53.239,-47.131,179.059,6.201,149.398
C01195=1133.047,-52.990,-47.142,179.060,6.201,149.397
C01196=1133.042,-52.740,-47.153,179.062,6.202,149.397
C01197=1133.037,-52.489,-47.164,179.065,6.202,149.396
C01198=1133.031,-52.240,-47.175,179.067,6.203,149.395
C01199=1133.026,-51.990,-47.185,179.069,6.203,149.395
C01200=1133.021,-51.741,-47.196,179.072,6.204,149.395
C01201=1133.016,-51.491,-47.207,179.074,6.205,149.394
C01202=1133.010,-51.221,-47.219,179.077,6.205,149.393
C01203=1133.004,-50.950,-47.231,179.079,6.206,149.393
C01204=1132.999,-50.679,-47.243,179.081,6.207,149.392
C01205=1132.993,-50.408,-47.254,179.084,6.207,149.392
C01206=1132.987,-50.158,-47.266,179.086,6.208,149.391
C01207=1132.982,-49.909,-47.276,179.088,6.208,149.390
C01208=1132.977,-49.659,-47.287,179.091,6.209,149.390
C01209=1132.972,-49.409,-47.298,179.093,6.210,149.390
C01210=1132.966,-49.160,-47.309,179.095,6.210,149.389
C01211=1132.961,-48.909,-47.320,179.098,6.211,149.388
C01212=1132.956,-48.660,-47.331,179.100,6.212,149.388
C01213=1132.951,-48.411,-47.342,179.102,6.213,149.387
C01214=1132.945,-48.160,-47.353,179.105,6.213,149.387
C01215=1132.940,-47.911,-47.364,179.107,6.214,149.386
C01216=1132.935,-47.661,-47.375,179.109,6.215,149.386
C01217=1132.929,-47.412,-47.386,179.111,6.215,149.385
C01218=1132.924,-47.162,-47.397,179.113,6.215,149.385
C01219=1132.919,-46.912,-47.408,179.116,6.216,149.384
C01220=1132.914,-46.663,-47.419,179.118,6.217,149.384
C01221=1132.908,-46.413,-47.430,179.120,6.217,149.383
C01222=1132.903,-46.164,-47.441,179.123,6.218,149.382
C01223=1132.898,-45.913,-47.452,179.125,6.218,149.382
C01224=1132.893,-45.663,-47.464,179.127,6.219,149.381
C01225=1132.887,-45.415,-47.474,179.129,6.220,149.381
C01226=1132.882,-45.164,-47.485,179.132,6.220,149.380
C01227=1132.877,-44.914,-47.497,179.134,6.221,149.380
C01228=1132.872,-44.665,-47.508,179.136,6.222,149.379
C01229=1132.867,-44.415,-47.518,179.138,6.223,149.379
C01230=1132.861,-44.165,-47.530,179.141,6.223,149.378
C01231=1132.856,-43.916,-47.541,179.143,6.224,149.378
C01232=1132.850,-43.666,-47.553,179.145,6.225,149.377
C01233=1132.845,-43.416,-47.564,179.148,6.225,149.376
C01234=1132.840,-43.167,-47.575,179.150,6.226,149.376
C01235=1132.835,-42.917,-47.586,179.152,6.227,149.376
C01236=1132.830,-42.667,-47.597,179.155,6.227,149.375
C01237=1132.824,-42.418,-47.608,179.157,6.228,149.374
C01238=1132.819,-42.168,-47.620,179.160,6.229,149.374
C01239=1132.814,-41.919,-47.631,179.161,6.229,149.373
C01240=1132.809,-41.668,-47.642,179.163,6.229,149.373
C01241=1132.803,-41.419,-47.653,179.166,6.230,149.372
C01242=1132.798,-41.169,-47.665,179.168,6.230,149.372
C01243=1132.793,-40.919,-47.676,179.170,6.231,149.371
C01244=1132.788,-40.671,-47.687,179.173,6.232,149.371
C01245=1132.782,-40.420,-47.699,179.175,6.232,149.370
C01246=1132.777,-40.170,-47.710,179.177,6.233,149.370
C01247=1132.772,-39.920,-47.722,179.180,6.234,149.369
C01248=1132.767,-39.672,-47.733,179.182,6.234,149.368
C01249=1132.761,-39.422,-47.744,179.184,6.235,149.368
C01250=1132.756,-39.171,-47.755,179.187,6.236,149.367
C01251=1132.750,-38.922,-47.767,179.189,6.237,149.367
C01252=1132.746,-38.672,-47.778,179.191,6.237,149.366
C01253=1132.740,-38.423,-47.790,179.194,6.238,149.366
C01254=1132.735,-38.173,-47.801,179.196,6.239,149.365
C01255=1132.729,-37.924,-47.813,179.198,6.239,149.365
C01256=1132.725,-37.674,-47.824,179.201,6.240,149.364
C01257=1132.719,-37.424,-47.836,179.203,6.241,149.364
C01258=1132.714,-37.174,-47.846,179.205,6.241,149.363
C01259=1132.708,-36.925,-47.858,179.208,6.242,149.363
C01260=1132.704,-36.675,-47.869,179.210,6.242,149.362
C01261=1132.698,-36.425,-47.881,179.212,6.243,149.362
C01262=1132.693,-36.175,-47.892,179.215,6.244,149.361
C01263=1132.688,-35.926,-47.904,179.217,6.244,149.360
C01264=1132.683,-35.677,-47.915,179.219,6.245,149.360
C01265=1132.677,-35.427,-47.927,179.221,6.246,149.359
C01266=1132.672,-35.177,-47.939,179.224,6.246,149.359
C01267=1132.667,-34.927,-47.950,179.226,6.247,149.358
C01268=1132.662,-34.677,-47.962,179.228,6.248,149.358
C01269=1132.656,-34.428,-47.973,179.231,6.248,149.357
C01270=1132.651,-34.178,-47.985,179.233,6.249,149.357
C01271=1132.646,-33.928,-47.997,179.235,6.250,149.356
C01272=1132.641,-33.679,-48.008,179.238,6.251,149.356
C01273=1132.635,-33.429,-48.020,179.241,6.252,149.355
C01274=1132.630,-33.180,-48.031,179.243,6.253,149.354
C01275=1132.625,-32.930,-48.043,179.245,6.253,149.354
C01276=1132.619,-32.680,-48.055,179.248,6.254,149.353
C01277=1132.615,-32.430,-48.066,179.250,6.255,149.353
C01278=1132.609,-32.180,-48.078,179.252,6.255,149.352
C01279=1132.604,-31.931,-48.089,179.254,6.256,149.352
C01280=1132.599,-31.681,-48.101,179.257,6.257,149.351
C01281=1132.593,-31.432,-48.112,179.259,6.257,149.351
C01282=1132.589,-31.183,-48.124,179.262,6.258,149.350
C01283=1132.583,-30.933,-48.136,179.264,6.259,149.350
C01284=1132.578,-30.683,-48.148,179.266,6.259,149.349
C01285=1132.573,-30.433,-48.160,179.269,6.260,149.349
C01286=1132.568,-30.183,-48.171,179.271,6.261,149.348
C01287=1132.562,-29.933,-48.183,179.273,6.261,149.347
C01288=1132.557,-29.684,-48.194,179.276,6.262,149.347
C01289=1132.552,-29.434,-48.206,179.278,6.263,149.346
C01290=1132.546,-29.185,-48.219,179.280,6.263,149.346
C01291=1132.542,-28.935,-48.230,179.283,6.264,149.345
C01292=1132.536,-28.686,-48.242,179.285,6.265,149.345
C01293=1132.531,-28.436,-48.254,179.287,6.265,149.344
C01294=1132.525,-28.186,-48.266,179.290,6.266,149.344
C01295=1132.521,-27.937,-48.278,179.292,6.267,149.343
C01296=1132.516,-27.687,-48.290,179.295,6.268,149.343
C01297=1132.510,-27.437,-48.301,179.297,6.269,149.342
C01298=1132.505,-27.187,-48.313,179.299,6.270,149.342
C01299=1132.500,-26.937,-48.325,179.302,6.270,149.341
C01300=1132.494,-26.689,-48.337,179.304,6.271,149.340
C01301=1132.489,-26.439,-48.349,179.307,6.271,149.340
C01302=1132.484,-26.189,-48.360,179.309,6.272,149.339
C01303=1132.479,-25.939,-48.372,179.311,6.273,149.339
C01304=1132.474,-25.690,-48.385,179.314,6.273,149.338
C01305=1132.468,-25.440,-48.396,179.316,6.274,149.338
C01306=1132.463,-25.169,-48.409,179.318,6.275,149.337
C01307=1132.457,-24.900,-48.422,179.321,6.276,149.337
C01308=1132.452,-24.629,-48.435,179.324,6.277,149.336
C01309=1132.446,-24.359,-48.448,179.326,6.277,149.335
C01310=1132.441,-24.109,-48.460,179.328,6.278,149.335
C01311=1132.436,-23.860,-48.472,179.331,6.279,149.334
C01312=1132.430,-23.610,-48.484,179.333,6.279,149.334
C01313=1132.425,-23.360,-48.496,179.336,6.281,149.333
C01314=1132.420,-23.111,-48.509,179.339,6.281,149.333
C01315=1132.415,-22.861,-48.520,179.341,6.282,149.332
C01316=1132.410,-22.612,-48.533,179.343,6.283,149.332
C01317=1132.405,-22.362,-48.545,179.345,6.284,149.331
C01318=1132.399,-22.112,-48.556,179.348,6.284,149.330
C01319=1132.394,-21.863,-48.569,179.350,6.285,149.330
C01320=1132.389,-21.613,-48.581,179.352,6.286,149.330
C01321=1132.383,-21.363,-48.594,179.355,6.286,149.329
C01322=1132.378,-21.113,-48.605,179.357,6.287,149.328
C01323=1132.373,-20.864,-48.617,179.360,6.288,149.328
C01324=1132.368,-20.614,-48.629,179.362,6.289,149.327
C01325=1132.363,-20.364,-48.641,179.365,6.290,149.327
C01326=1132.358,-20.115,-48.654,179.367,6.290,149.326
C01327=1132.352,-19.865,-48.666,179.369,6.291,149.326
C01328=1132.347,-19.616,-48.678,179.372,6.292,149.325
C01329=1132.342,-19.366,-48.690,179.374,6.292,149.325
C01330=1132.337,-19.117,-48.703,179.376,6.293,149.324
C01331=1132.331,-18.867,-48.715,179.379,6.294,149.323
C01332=1132.326,-18.617,-48.727,179.381,6.295,149.323
C01333=1132.321,-18.367,-48.739,179.384,6.296,149.323
C01334=1132.315,-18.118,-48.752,179.386,6.296,149.322
C01335=1132.310,-17.868,-48.764,179.388,6.297,149.321
C01336=1132.305,-17.619,-48.776,179.391,6.298,149.321
C01337=1132.299,-17.369,-48.788,179.393,6.298,149.320
C01338=1132.294,-17.120,-48.801,179.395,6.299,149.320
C01339=1132.289,-16.870,-48.813,179.398,6.300,149.319
C01340=1132.284,-16.620,-48.825,179.401,6.301,149.319
C01341=1132.279,-16.370,-48.838,179.403,6.302,149.318
C01342=1132.274,-16.120,-48.850,179.405,6.303,149.318
C01343=1132.269,-15.871,-48.863,179.407,6.303,149.317
C01344=1132.263,-15.621,-48.875,179.410,6.304,149.316
C01345=1132.258,-15.372,-48.887,179.412,6.305,149.316
C01346=1132.253,-15.123,-48.900,179.414,6.305,149.316
C01347=1132.248,-14.873,-48.912,179.418,6.307,149.315
C01348=1132.243,-14.623,-48.924,179.420,6.307,149.314
C01349=1132.237,-14.373,-48.936,179.422,6.308,149.314
C01350=1132.233,-14.123,-48.949,179.425,6.309,149.313
C01351=1132.227,-13.874,-48.962,179.427,6.309,149.313
C01352=1132.222,-13.624,-48.974,179.429,6.310,149.312
C01353=1132.217,-13.375,-48.986,179.432,6.311,149.312
C01354=1132.212,-13.125,-48.999,179.435,6.312,149.311
C01355=1132.207,-12.876,-49.011,179.437,6.313,149.311
C01356=1132.201,-12.626,-49.023,179.439,6.313,149.310
C01357=1132.197,-12.376,-49.036,179.442,6.314,149.309
C01358=1132.192,-12.127,-49.049,179.444,6.315,149.309
C01359=1132.186,-11.877,-49.061,179.446,6.316,149.309
C01360=1132.180,-11.627,-49.074,179.449,6.317,149.308
C01361=1132.175,-11.378,-49.086,179.451,6.318,149.307
C01362=1132.171,-11.128,-49.099,179.454,6.319,149.307
C01363=1132.165,-10.878,-49.111,179.456,6.319,149.306
C01364=1132.160,-10.629,-49.124,179.458,6.320,149.306
C01365=1132.155,-10.379,-49.137,179.461,6.321,149.305
C01366=1132.150,-10.130,-49.149,179.464,6.322,149.305
C01367=1132.145,-9.881,-49.162,179.466,6.323,149.304
C01368=1132.139,-9.630,-49.175,179.468,6.323,149.304
C01369=1132.134,-9.380,-49.187,179.471,6.324,149.303
C01370=1132.129,-9.131,-49.200,179.473,6.325,149.302
C01371=1132.124,-8.882,-49.212,179.476,6.326,149.302
C01372=1132.119,-8.632,-49.225,179.479,6.327,149.301
C01373=1132.114,-8.382,-49.238,179.481,6.327,149.301
C01374=1132.108,-8.132,-49.250,179.483,6.328,149.300
C01375=1132.103,-7.883,-49.263,179.486,6.329,149.300
C01376=1132.098,-7.634,-49.276,179.488,6.330,149.299
C01377=1132.093,-7.384,-49.289,179.490,6.331,149.299
C01378=1132.088,-7.134,-49.301,179.493,6.332,149.298
C01379=1132.082,-6.885,-49.314,179.495,6.332,149.298
C01380=1132.077,-6.635,-49.327,179.498,6.333,149.297
C01381=1132.073,-6.385,-49.340,179.500,6.335,149.297
C01382=1132.067,-6.136,-49.353,179.503,6.335,149.296
C01383=1132.062,-5.886,-49.366,179.505,6.336,149.295
C01384=1132.056,-5.636,-49.378,179.507,6.337,149.295
C01385=1132.052,-5.386,-49.391,179.510,6.337,149.294
C01386=1132.046,-5.137,-49.403,179.513,6.339,149.294
C01387=1132.041,-4.887,-49.416,179.515,6.339,149.293
C01388=1132.036,-4.637,-49.429,179.518,6.340,149.293
C01389=1132.031,-4.388,-49.442,179.520,6.341,149.292
C01390=1132.026,-4.139,-49.455,179.522,6.341,149.292
C01391=1132.020,-3.889,-49.468,179.525,6.343,149.291
C01392=1132.015,-3.639,-49.481,179.527,6.343,149.291
C01393=1132.010,-3.390,-49.493,179.530,6.344,149.290
C01394=1132.004,-3.140,-49.507,179.532,6.345,149.289
C01395=1132.000,-2.890,-49.519,179.535,6.346,149.289
C01396=1131.995,-2.641,-49.532,179.537,6.347,149.288
C01397=1131.989,-2.392,-49.546,179.540,6.347,149.288
C01398=1131.985,-2.142,-49.559,179.542,6.348,149.287
C01399=1131.980,-1.893,-49.572,179.544,6.349,149.287
C01400=1131.974,-1.643,-49.585,179.547,6.351,149.286
C01401=1131.969,-1.393,-49.598,179.550,6.351,149.286
C01402=1131.964,-1.144,-49.610,179.552,6.352,149.285
C01403=1131.958,-0.894,-49.624,179.554,6.353,149.285
C01404=1131.954,-0.644,-49.636,179.557,6.354,149.284
C01405=1131.948,-0.394,-49.650,179.559,6.355,149.284
C01406=1131.943,-0.145,-49.662,179.562,6.355,149.283
C01407=1131.939,0.104,-49.676,179.564,6.356,149.282
C01408=1131.933,0.354,-49.689,179.567,6.357,149.282
C01409=1131.928,0.603,-49.702,179.569,6.358,149.282
C01410=1131.922,0.873,-49.716,179.572,6.359,149.281
C01411=1131.917,1.143,-49.730,179.575,6.360,149.280
C01412=1131.911,1.413,-49.745,179.577,6.361,149.280
C01413=1131.905,1.682,-49.759,179.580,6.362,149.279
C01414=1131.901,1.932,-49.772,179.583,6.363,149.279
C01415=1131.895,2.181,-49.786,179.585,6.363,149.278
C01416=1131.890,2.430,-49.798,179.587,6.364,149.278
C01417=1131.885,2.681,-49.812,179.590,6.365,149.277
C01418=1131.879,2.930,-49.824,179.593,6.366,149.276
C01419=1131.875,3.180,-49.837,179.595,6.367,149.276
C01420=1131.869,3.429,-49.851,179.597,6.367,149.275
C01421=1131.864,3.678,-49.864,179.600,6.369,149.275
C01422=1131.859,3.929,-49.877,179.602,6.370,149.274
C01423=1131.854,4.177,-49.891,179.605,6.370,149.274
C01424=1131.849,4.428,-49.904,179.608,6.372,149.273
C01425=1131.844,4.677,-49.917,179.610,6.373,149.273
C01426=1131.839,4.927,-49.930,179.613,6.373,149.272
C01427=1131.834,5.176,-49.944,179.615,6.374,149.272
C01428=1131.828,5.426,-49.957,179.618,6.376,149.271
C01429=1131.823,5.676,-49.970,179.620,6.376,149.271
C01430=1131.818,5.925,-49.984,179.622,6.377,149.270
C01431=1131.813,6.175,-49.997,179.625,6.378,149.270
C01432=1131.808,6.424,-50.011,179.627,6.379,149.269
C01433=1131.802,6.674,-50.024,179.630,6.380,149.268
C01434=1131.797,6.923,-50.037,179.632,6.380,149.268
C01435=1131.792,7.173,-50.051,179.635,6.382,149.267
C01436=1131.787,7.422,-50.064,179.638,6.382,149.267
C01437=1131.782,7.673,-50.077,179.640,6.383,149.266
C01438=1131.777,7.921,-50.091,179.643,6.385,149.266
C01439=1131.772,8.172,-50.104,179.645,6.385,149.265
C01440=1131.766,8.421,-50.118,179.647,6.386,149.265
C01441=1131.762,8.671,-50.131,179.650,6.387,149.264
C01442=1131.756,8.920,-50.145,179.653,6.388,149.264
C01443=1131.751,9.170,-50.158,179.655,6.389,149.263
C01444=1131.746,9.419,-50.172,179.657,6.390,149.263
C01445=1131.741,9.669,-50.185,179.660,6.391,149.262
C01446=1131.736,9.918,-50.199,179.663,6.392,149.261
C01447=1131.731,10.168,-50.212,179.665,6.392,149.261
C01448=1131.725,10.417,-50.226,179.668,6.394,149.260
C01449=1131.721,10.667,-50.239,179.670,6.394,149.260
C01450=1131.715,10.916,-50.253,179.672,6.395,149.259
C01451=1131.710,11.166,-50.267,179.675,6.397,149.259
C01452=1131.706,11.416,-50.280,179.678,6.397,149.258
C01453=1131.700,11.665,-50.293,179.680,6.398,149.258
C01454=1131.695,11.915,-50.308,179.683,6.400,149.257
C01455=1131.690,12.164,-50.320,179.685,6.400,149.257
C01456=1131.685,12.414,-50.335,179.688,6.401,149.256
C01457=1131.679,12.663,-50.349,179.690,6.403,149.256
C01458=1131.674,12.914,-50.362,179.693,6.403,149.255
C01459=1131.670,13.163,-50.376,179.695,6.404,149.255
C01460=1131.664,13.413,-50.389,179.698,6.405,149.254
C01461=1131.659,13.662,-50.403,179.701,6.406,149.253
C01462=1131.653,13.911,-50.417,179.703,6.407,149.253
C01463=1131.649,14.161,-50.430,179.706,6.408,149.253
C01464=1131.644,14.411,-50.444,179.708,6.409,149.252
C01465=1131.638,14.660,-50.458,179.710,6.409,149.251
C01466=1131.633,14.910,-50.472,179.713,6.411,149.251
C01467=1131.628,15.159,-50.485,179.716,6.412,149.250
C01468=1131.623,15.409,-50.499,179.718,6.412,149.250
C01469=1131.618,15.659,-50.513,179.721,6.414,149.249
C01470=1131.613,15.908,-50.527,179.723,6.414,149.249
C01471=1131.608,16.158,-50.541,179.726,6.415,149.248
C01472=1131.602,16.407,-50.554,179.728,6.417,149.248
C01473=1131.598,16.657,-50.568,179.731,6.418,149.247
C01474=1131.593,16.907,-50.582,179.734,6.419,149.247
C01475=1131.587,17.156,-50.596,179.736,6.420,149.246
C01476=1131.582,17.406,-50.610,179.738,6.420,149.246
C01477=1131.578,17.655,-50.624,179.741,6.422,149.245
C01478=1131.572,17.904,-50.637,179.744,6.422,149.244
C01479=1131.567,18.154,-50.652,179.746,6.423,149.244
C01480=1131.562,18.404,-50.666,179.749,6.424,149.243
C01481=1131.556,18.653,-50.679,179.751,6.425,149.243
C01482=1131.551,18.903,-50.693,179.753,6.426,149.242
C01483=1131.546,19.153,-50.708,179.757,6.427,149.242
C01484=1131.541,19.401,-50.721,179.759,6.428,149.241
C01485=1131.537,19.651,-50.735,179.762,6.430,149.241
C01486=1131.532,19.901,-50.750,179.764,6.430,149.240
C01487=1131.526,20.151,-50.763,179.766,6.431,149.240
C01488=1131.521,20.400,-50.777,179.769,6.433,149.239
C01489=1131.516,20.650,-50.791,179.771,6.433,149.239
C01490=1131.511,20.900,-50.806,179.775,6.435,149.238
C01491=1131.505,21.149,-50.820,179.777,6.435,149.238
C01492=1131.500,21.398,-50.834,179.779,6.436,149.237
C01493=1131.495,21.648,-50.848,179.782,6.437,149.236
C01494=1131.490,21.898,-50.862,179.784,6.438,149.236
C01495=1131.486,22.146,-50.876,179.787,6.440,149.236
C01496=1131.481,22.396,-50.890,179.790,6.440,149.235
C01497=1131.475,22.647,-50.904,179.792,6.441,149.234
C01498=1131.470,22.896,-50.918,179.795,6.443,149.234
C01499=1131.465,23.145,-50.932,179.797,6.443,149.233
C01500=1131.460,23.395,-50.946,179.800,6.445,149.233
C01501=1131.455,23.645,-50.960,179.802,6.446,149.232
C01502=1131.450,23.894,-50.975,179.804,6.446,149.232
C01503=1131.444,24.143,-50.988,179.808,6.448,149.231
C01504=1131.439,24.393,-51.003,179.810,6.448,149.231
C01505=1131.435,24.643,-51.017,179.813,6.450,149.230
C01506=1131.430,24.893,-51.031,179.815,6.451,149.230
C01507=1131.424,25.141,-51.046,179.817,6.451,149.229
C01508=1131.419,25.391,-51.060,179.820,6.453,149.229
C01509=1131.414,25.640,-51.074,179.823,6.453,149.228
C01510=1131.409,25.890,-51.089,179.826,6.455,149.228
C01511=1131.404,26.140,-51.104,179.828,6.456,149.227
C01512=1131.398,26.389,-51.118,179.831,6.457,149.226
C01513=1131.393,26.639,-51.132,179.833,6.458,149.226
C01514=1131.388,26.908,-51.148,179.836,6.459,149.226
C01515=1131.383,27.177,-51.162,179.839,6.460,149.225
C01516=1131.378,27.446,-51.178,179.841,6.462,149.224
C01517=1131.372,27.715,-51.193,179.845,6.463,149.224
C01518=1131.366,27.965,-51.208,179.847,6.464,149.223
C01519=1131.361,28.214,-51.223,179.849,6.464,149.223
C01520=1131.356,28.463,-51.237,179.852,6.466,149.222
C01521=1131.351,28.713,-51.251,179.854,6.466,149.222
C01522=1131.346,28.963,-51.266,179.857,6.468,149.221
C01523=1131.341,29.212,-51.280,179.860,6.468,149.221
C01524=1131.337,29.462,-51.295,179.863,6.470,149.220
C01525=1131.331,29.711,-51.309,179.865,6.471,149.220
C01526=1131.325,29.961,-51.324,179.868,6.472,149.219
C01527=1131.321,30.210,-51.338,179.870,6.473,149.219
C01528=1131.316,30.460,-51.352,179.872,6.474,149.218
C01529=1131.311,30.709,-51.367,179.875,6.475,149.218
C01530=1131.306,30.959,-51.381,179.878,6.476,149.217
C01531=1131.301,31.209,-51.396,179.881,6.477,149.216
C01532=1131.296,31.458,-51.411,179.883,6.478,149.216
C01533=1131.291,31.708,-51.426,179.886,6.480,149.215
C01534=1131.285,31.957,-51.439,179.888,6.480,149.215
C01535=1131.280,32.206,-51.454,179.891,6.482,149.214
C01536=1131.276,32.455,-51.469,179.894,6.482,149.214
C01537=1131.270,32.705,-51.484,179.896,6.484,149.213
C01538=1131.265,32.955,-51.498,179.898,6.485,149.213
C01539=1131.260,33.204,-51.513,179.901,6.486,149.212
C01540=1131.255,33.454,-51.527,179.904,6.487,149.212
C01541=1131.250,33.704,-51.542,179.907,6.489,149.211
C01542=1131.245,33.953,-51.557,179.909,6.489,149.211
C01543=1131.240,34.203,-51.571,179.912,6.491,149.210
C01544=1131.235,34.452,-51.586,179.914,6.491,149.210
C01545=1131.230,34.702,-51.601,179.917,6.493,149.209
C01546=1131.225,34.952,-51.615,179.919,6.494,149.209
C01547=1131.220,35.201,-51.630,179.922,6.495,149.208
C01548=1131.214,35.451,-51.645,179.925,6.496,149.208
C01549=1131.210,35.700,-51.660,179.927,6.498,149.207
C01550=1131.205,35.950,-51.675,179.930,6.498,149.207
C01551=1131.199,36.199,-51.690,179.933,6.500,149.206
C01552=1131.194,36.448,-51.704,179.935,6.500,149.206
C01553=1131.189,36.697,-51.719,179.938,6.502,149.205
C01554=1131.183,36.947,-51.734,179.940,6.502,149.205
C01555=1131.179,37.196,-51.749,179.943,6.504,149.204
C01556=1131.174,37.446,-51.763,179.945,6.505,149.204
C01557=1131.168,37.695,-51.779,179.949,6.506,149.203
C01558=1131.163,37.945,-51.793,179.951,6.507,149.202
C01559=1131.159,38.194,-51.808,179.953,6.509,149.202
C01560=1131.154,38.445,-51.823,179.956,6.509,149.201
C01561=1131.149,38.694,-51.838,179.959,6.511,149.201
C01562=1131.143,38.944,-51.853,179.961,6.511,149.200
C01563=1131.139,39.193,-51.868,179.964,6.513,149.200
C01564=1131.134,39.442,-51.883,179.966,6.514,149.199
C01565=1131.128,39.692,-51.898,179.969,6.515,149.199
C01566=1131.124,39.941,-51.913,179.971,6.516,149.198
C01567=1131.118,40.191,-51.928,179.975,6.517,149.198
C01568=1131.113,40.440,-51.943,179.977,6.518,149.197
C01569=1131.108,40.690,-51.958,179.980,6.520,149.197
C01570=1131.103,40.939,-51.973,179.982,6.520,149.196
C01571=1131.098,41.189,-51.988,179.985,6.522,149.196
C01572=1131.093,41.438,-52.003,179.987,6.523,149.195
C01573=1131.088,41.688,-52.018,179.990,6.524,149.195
C01574=1131.083,41.937,-52.033,179.993,6.525,149.194
C01575=1131.078,42.186,-52.048,179.995,6.526,149.194
C01576=1131.072,42.436,-52.063,179.998,6.528,149.193
C01577=1131.068,42.685,-52.078,-180.000,6.529,149.193
C01578=1131.063,42.935,-52.094,-179.997,6.530,149.192
C01579=1131.058,43.185,-52.108,-179.994,6.531,149.192
C01580=1131.053,43.434,-52.124,-179.992,6.532,149.191
C01581=1131.048,43.684,-52.139,-179.989,6.533,149.191
C01582=1131.043,43.933,-52.154,-179.986,6.534,149.190
C01583=1131.038,44.183,-52.169,-179.983,6.536,149.190
C01584=1131.032,44.432,-52.184,-179.981,6.537,149.189
C01585=1131.027,44.681,-52.200,-179.978,6.538,149.189
C01586=1131.023,44.931,-52.215,-179.976,6.539,149.188
C01587=1131.017,45.181,-52.231,-179.973,6.541,149.188
C01588=1131.012,45.430,-52.245,-179.971,6.541,149.187
C01589=1131.007,45.680,-52.261,-179.968,6.543,149.187
C01590=1131.002,45.929,-52.276,-179.965,6.544,149.186
C01591=1130.997,46.178,-52.291,-179.963,6.545,149.186
C01592=1130.992,46.428,-52.307,-179.960,6.546,149.185
C01593=1130.988,46.677,-52.322,-179.957,6.547,149.185
C01594=1130.982,46.927,-52.338,-179.955,6.549,149.184
C01595=1130.977,47.177,-52.352,-179.952,6.550,149.184
C01596=1130.972,47.426,-52.368,-179.949,6.551,149.183
C01597=1130.966,47.675,-52.383,-179.946,6.553,149.183
C01598=1130.962,47.925,-52.399,-179.944,6.553,149.182
C01599=1130.957,48.175,-52.414,-179.941,6.555,149.182
C01600=1130.952,48.424,-52.430,-179.939,6.555,149.181
C01601=1130.947,48.673,-52.445,-179.936,6.557,149.181
C01602=1130.942,48.922,-52.460,-179.933,6.559,149.180
C01603=1130.937,49.173,-52.476,-179.931,6.560,149.180
C01604=1130.932,49.422,-52.491,-179.928,6.561,149.179
C01605=1130.927,49.671,-52.507,-179.926,6.562,149.179
C01606=1130.921,49.920,-52.523,-179.923,6.563,149.178
C01607=1130.917,50.170,-52.538,-179.920,6.565,149.177
C01608=1130.912,50.420,-52.553,-179.918,6.565,149.177
C01609=1130.907,50.669,-52.569,-179.915,6.567,149.177
C01610=1130.902,50.918,-52.584,-179.913,6.568,149.176
C01611=1130.897,51.168,-52.600,-179.909,6.569,149.175
C01612=1130.892,51.418,-52.616,-179.907,6.571,149.175
C01613=1130.886,51.667,-52.631,-179.905,6.572,149.175
C01614=1130.882,51.916,-52.646,-179.902,6.573,149.174
C01615=1130.877,52.166,-52.662,-179.899,6.574,149.173
C01616=1130.872,52.416,-52.678,-179.896,6.575,149.173
C01617=1130.866,52.665,-52.693,-179.894,6.577,149.173
C01618=1130.861,52.933,-52.710,-179.891,6.577,149.172
C01619=1130.856,53.202,-52.727,-179.888,6.579,149.171
C01620=1130.851,53.471,-52.744,-179.885,6.581,149.171
C01621=1130.845,53.739,-52.761,-179.882,6.582,149.170
C01622=1130.840,53.989,-52.777,-179.879,6.583,149.170
C01623=1130.834,54.238,-52.792,-179.877,6.584,149.169
C01624=1130.830,54.488,-52.808,-179.874,6.586,149.169
C01625=1130.825,54.737,-52.823,-179.871,6.587,149.168
C01626=1130.820,54.986,-52.840,-179.869,6.588,149.168
C01627=1130.815,55.236,-52.856,-179.866,6.590,149.167
C01628=1130.810,55.486,-52.871,-179.864,6.590,149.167
C01629=1130.804,55.735,-52.887,-179.861,6.592,149.166
C01630=1130.801,55.984,-52.903,-179.858,6.593,149.166
C01631=1130.795,56.234,-52.918,-179.856,6.594,149.165
C01632=1130.790,56.483,-52.934,-179.853,6.595,149.165
C01633=1130.785,56.733,-52.950,-179.850,6.597,149.164
C01634=1130.780,56.982,-52.966,-179.848,6.598,149.164
C01635=1130.775,57.231,-52.982,-179.845,6.600,149.163
C01636=1130.770,57.481,-52.998,-179.842,6.601,149.163
C01637=1130.764,57.731,-53.013,-179.840,6.602,149.162
C01638=1130.759,57.980,-53.030,-179.837,6.603,149.162
C01639=1130.755,58.230,-53.046,-179.834,6.605,149.161
C01640=1130.750,58.479,-53.061,-179.832,6.605,149.161
C01641=1130.745,58.728,-53.077,-179.829,6.607,149.160
C01642=1130.738,59.073,-53.099,-179.825,6.609,149.160
C01643=1130.712,60.364,-53.184,179.810,7.354,149.432
C01644=1130.707,60.613,-53.201,179.812,7.358,149.432
C01645=1130.702,60.863,-53.217,179.813,7.362,149.433
C01646=1130.697,61.112,-53.233,179.815,7.366,149.433
C01647=1130.693,61.340,-53.248,179.815,7.369,149.434
C01648=1130.688,61.569,-53.263,179.817,7.373,149.434
C01649=1130.684,61.799,-53.278,179.819,7.377,149.435
C01650=1130.679,62.027,-53.293,179.820,7.380,149.435
C01651=1130.675,62.256,-53.308,179.821,7.384,149.436
C01652=1130.670,62.485,-53.322,179.822,7.388,149.436
C01653=1130.666,62.713,-53.337,179.823,7.391,149.437
C01654=1130.660,62.942,-53.353,179.825,7.395,149.437
C01655=1130.656,63.191,-53.369,179.826,7.399,149.437
C01656=1130.651,63.441,-53.385,179.827,7.404,149.438
C01657=1130.646,63.690,-53.402,179.829,7.407,149.438
C01658=1130.642,63.940,-53.418,179.831,7.411,149.439
C01659=1130.636,64.189,-53.435,179.832,7.416,149.439
C01660=1130.631,64.439,-53.451,179.833,7.420,149.440
C01661=1130.626,64.688,-53.467,179.835,7.423,149.440
C01662=1130.621,64.937,-53.484,179.836,7.428,149.441
C01663=1130.617,65.187,-53.501,179.837,7.432,149.441
C01664=1130.611,65.436,-53.517,179.839,7.436,149.442
C01665=1130.606,65.686,-53.534,179.841,7.439,149.442
C01666=1130.601,65.935,-53.550,179.842,7.444,149.443
C01667=1130.597,66.184,-53.567,179.843,7.448,149.443
C01668=1130.592,66.434,-53.584,179.845,7.452,149.444
C01669=1130.586,66.683,-53.599,179.846,7.456,149.444
C01670=1130.582,66.933,-53.616,179.848,7.460,149.445
C01671=1130.577,67.182,-53.633,179.849,7.464,149.445
C01672=1130.571,67.431,-53.650,179.851,7.468,149.446
C01673=1130.567,67.681,-53.666,179.852,7.472,149.446
C01674=1130.562,67.930,-53.683,179.853,7.476,149.447
C01675=1130.557,68.179,-53.700,179.855,7.480,149.447
C01676=1130.552,68.429,-53.717,179.856,7.484,149.448
C01677=1130.547,68.678,-53.733,179.858,7.488,149.448
C01678=1130.542,68.928,-53.749,179.859,7.492,149.449
C01679=1130.537,69.178,-53.766,179.861,7.496,149.449
C01680=1130.532,69.426,-53.782,179.862,7.500,149.450
C01681=1130.527,69.676,-53.800,179.863,7.504,149.450
C01682=1130.522,69.926,-53.816,179.865,7.508,149.451
C01683=1130.517,70.174,-53.833,179.867,7.512,149.451
C01684=1130.512,70.424,-53.850,179.868,7.516,149.452
C01685=1130.508,70.674,-53.867,179.869,7.520,149.452
C01686=1130.502,70.923,-53.884,179.871,7.524,149.452
C01687=1130.497,71.172,-53.900,179.872,7.528,149.453
C01688=1130.493,71.422,-53.917,179.874,7.532,149.454
C01689=1130.488,71.672,-53.934,179.875,7.536,149.454
C01690=1130.482,71.920,-53.950,179.877,7.540,149.454
C01691=1130.478,72.169,-53.968,179.878,7.543,149.455
C01692=1130.473,72.419,-53.985,179.879,7.547,149.455
C01693=1130.468,72.669,-54.002,179.880,7.551,149.456
C01694=1130.463,72.918,-54.019,179.882,7.555,149.456
C01695=1130.458,73.167,-54.035,179.884,7.559,149.457
C01696=1130.453,73.417,-54.052,179.885,7.563,149.457
C01697=1130.449,73.666,-54.069,179.886,7.567,149.458
C01698=1130.443,73.915,-54.086,179.888,7.571,149.458
C01699=1130.439,74.164,-54.103,179.889,7.575,149.459
C01700=1130.433,74.414,-54.121,179.891,7.579,149.459
C01701=1130.429,74.664,-54.137,179.892,7.583,149.460
C01702=1130.423,74.913,-54.154,179.894,7.587,149.460
C01703=1130.419,75.128,-54.169,179.895,7.591,149.461
C01704=1130.415,75.343,-54.184,179.896,7.594,149.461
C01705=1130.411,75.558,-54.198,179.898,7.598,149.461
C01706=1130.406,75.773,-54.213,179.899,7.601,149.462
C01707=1130.402,75.988,-54.228,179.900,7.604,149.462
C01708=1130.398,76.203,-54.243,179.901,7.608,149.463
C01709=1130.393,76.419,-54.258,179.902,7.611,149.463
C01710=1130.389,76.634,-54.272,179.904,7.615,149.463
C01711=1130.385,76.883,-54.290,179.905,7.618,149.464
C01712=1130.380,77.133,-54.307,179.906,7.622,149.465
C01713=1130.375,77.382,-54.324,179.907,7.626,149.465
C01714=1130.369,77.631,-54.341,179.907,7.629,149.466
C01715=1130.364,77.880,-54.359,179.909,7.633,149.466
C01716=1130.360,78.130,-54.375,179.909,7.636,149.467
C01717=1130.355,78.380,-54.393,179.911,7.640,149.467
C01718=1130.351,78.628,-54.410,179.912,7.644,149.468
C01719=1130.345,78.878,-54.427,179.913,7.648,149.468
C01720=1130.340,79.127,-54.445,179.914,7.651,149.469
C01721=1130.335,79.376,-54.462,179.915,7.656,149.470
C01722=1130.330,79.626,-54.479,179.916,7.659,149.470
C01723=1130.325,79.875,-54.497,179.917,7.663,149.471
C01724=1130.321,80.125,-54.513,179.918,7.667,149.471
C01725=1130.316,80.374,-54.531,179.919,7.670,149.472
C01726=1130.311,80.624,-54.549,179.921,7.674,149.472
C01727=1130.306,80.873,-54.565,179.921,7.678,149.473
C01728=1130.301,81.122,-54.583,179.923,7.682,149.473
C01729=1130.295,81.371,-54.600,179.923,7.685,149.474
C01730=1130.291,81.620,-54.618,179.925,7.689,149.474
C01731=1130.286,81.870,-54.635,179.926,7.693,149.475
C01732=1130.281,82.119,-54.653,179.927,7.696,149.475
C01733=1130.276,82.369,-54.670,179.928,7.700,149.476
C01734=1130.272,82.618,-54.688,179.930,7.705,149.476
C01735=1130.266,82.868,-54.705,179.930,7.708,149.477
C01736=1130.262,83.117,-54.723,179.932,7.712,149.477
C01737=1130.257,83.366,-54.739,179.933,7.716,149.478
C01738=1130.252,83.615,-54.757,179.934,7.719,149.478
C01739=1130.247,83.865,-54.775,179.935,7.723,149.479
C01740=1130.242,84.114,-54.793,179.937,7.727,149.479
C01741=1130.237,84.364,-54.811,179.938,7.731,149.480
C01742=1130.233,84.613,-54.827,179.939,7.735,149.480
C01743=1130.228,84.862,-54.845,179.941,7.739,149.481
C01744=1130.222,85.112,-54.863,179.942,7.742,149.481
C01745=1130.218,85.361,-54.881,179.943,7.747,149.482
C01746=1130.212,85.610,-54.898,179.945,7.751,149.482
C01747=1130.208,85.859,-54.915,179.946,7.754,149.483
C01748=1130.203,86.108,-54.933,179.947,7.758,149.483
C01749=1130.197,86.358,-54.950,179.949,7.762,149.484
C01750=1130.193,86.607,-54.968,179.950,7.766,149.484
C01751=1130.188,86.857,-54.986,179.952,7.770,149.485
C01752=1130.183,87.106,-55.004,179.953,7.774,149.485
C01753=1130.178,87.355,-55.021,179.954,7.777,149.486
C01754=1130.173,87.604,-55.039,179.955,7.781,149.486
C01755=1130.168,87.854,-55.057,179.957,7.785,149.487
C01756=1130.163,88.103,-55.074,179.958,7.789,149.487
C01757=1130.159,88.353,-55.092,179.960,7.793,149.488
C01758=1130.154,88.602,-55.110,179.961,7.797,149.488
C01759=1130.150,88.817,-55.126,179.962,7.800,149.489
C01760=1130.145,89.032,-55.140,179.964,7.804,149.489
C01761=1130.141,89.247,-55.156,179.965,7.807,149.489
C01762=1130.137,89.462,-55.171,179.967,7.811,149.490
C01763=1130.132,89.677,-55.187,179.968,7.814,149.490
C01764=1130.128,89.892,-55.202,179.969,7.817,149.490
C01765=1130.124,90.108,-55.217,179.971,7.821,149.491
C01766=1130.120,90.322,-55.233,179.972,7.824,149.491
C01767=1130.115,90.572,-55.251,179.973,7.828,149.492
C01768=1130.110,90.821,-55.269,179.975,7.832,149.492
C01769=1130.105,91.070,-55.287,179.976,7.835,149.493
C01770=1130.101,91.319,-55.305,179.978,7.839,149.493
C01771=1130.095,91.569,-55.322,179.979,7.843,149.493
C01772=1130.090,91.818,-55.340,179.981,7.847,149.494
C01773=1130.085,92.067,-55.358,179.983,7.851,149.494
C01774=1130.081,92.317,-55.376,179.985,7.856,149.495
C01775=1130.076,92.566,-55.394,179.987,7.860,149.495
C01776=1130.071,92.816,-55.412,179.988,7.863,149.496
C01777=1130.066,93.065,-55.430,179.990,7.867,149.496
C01778=1130.062,93.314,-55.448,179.991,7.871,149.496
C01779=1130.057,93.563,-55.466,179.993,7.875,149.497
C01780=1130.052,93.812,-55.484,179.994,7.879,149.497
C01781=1130.047,94.061,-55.502,179.996,7.883,149.498
C01782=1130.042,94.311,-55.521,179.998,7.887,149.498
C01783=1130.038,94.561,-55.538,-180.000,7.891,149.498
C01784=1130.032,94.810,-55.557,-179.998,7.895,149.499
C01785=1130.027,95.059,-55.575,-179.996,7.899,149.499
C01786=1130.022,95.308,-55.593,-179.995,7.903,149.500
C01787=1130.017,95.558,-55.611,-179.993,7.907,149.500
C01788=1130.013,95.807,-55.629,-179.991,7.911,149.500
C01789=1130.008,96.057,-55.647,-179.989,7.915,149.501
C01790=1130.003,96.305,-55.666,-179.987,7.919,149.501
C01791=1129.998,96.554,-55.684,-179.986,7.923,149.502
C01792=1129.993,96.804,-55.703,-179.984,7.927,149.502
C01793=1129.988,97.054,-55.721,-179.981,7.931,149.502
C01794=1129.984,97.303,-55.739,-179.980,7.935,149.503
C01795=1129.979,97.552,-55.757,-179.978,7.939,149.503
C01796=1129.974,97.801,-55.775,-179.977,7.942,149.503
C01797=1129.968,98.050,-55.794,-179.974,7.947,149.504
C01798=1129.964,98.300,-55.812,-179.972,7.951,149.504
C01799=1129.959,98.549,-55.830,-179.971,7.955,149.505
C01800=1129.954,98.798,-55.848,-179.968,7.959,149.505
C01801=1129.950,99.047,-55.867,-179.966,7.963,149.505
C01802=1129.945,99.297,-55.886,-179.964,7.966,149.505
C01803=1129.940,99.546,-55.904,-179.962,7.971,149.506
C01804=1129.935,99.795,-55.922,-179.961,7.975,149.506
C01805=1129.931,100.045,-55.941,-179.959,7.978,149.506
C01806=1129.925,100.294,-55.960,-179.956,7.983,149.507
C01807=1129.920,100.543,-55.978,-179.954,7.986,149.507
C01808=1129.916,100.792,-55.996,-179.953,7.990,149.508
C01809=1129.911,101.042,-56.015,-179.950,7.995,149.508
C01810=1129.906,101.291,-56.033,-179.948,7.998,149.508
C01811=1129.901,101.540,-56.052,-179.946,8.003,149.508
C01812=1129.896,101.790,-56.071,-179.944,8.007,149.509
C01813=1129.891,102.039,-56.090,-179.941,8.011,149.509
C01814=1129.886,102.288,-56.108,-179.939,8.014,149.509
C01815=1129.882,102.503,-56.124,-179.938,8.018,149.510
C01816=1129.878,102.718,-56.140,-179.936,8.022,149.510
C01817=1129.874,102.933,-56.156,-179.934,8.025,149.510
C01818=1129.870,103.147,-56.172,-179.932,8.028,149.510
C01819=1129.865,103.362,-56.188,-179.930,8.032,149.511
C01820=1129.862,103.578,-56.204,-179.928,8.035,149.511
C01821=1129.857,103.792,-56.221,-179.926,8.039,149.511
C01822=1129.852,104.007,-56.237,-179.924,8.042,149.511
C01823=1129.848,104.257,-56.256,-179.922,8.046,149.512
C01824=1129.844,104.506,-56.274,-179.920,8.050,149.512
C01825=1129.838,104.755,-56.293,-179.918,8.054,149.512
C01826=1129.834,105.005,-56.312,-179.915,8.058,149.513
C01827=1129.829,105.253,-56.331,-179.913,8.062,149.513
C01828=1129.825,105.503,-56.350,-179.911,8.066,149.513
C01829=1129.819,105.752,-56.368,-179.909,8.070,149.513
C01830=1129.814,106.001,-56.387,-179.906,8.074,149.513
C01831=1129.809,106.251,-56.406,-179.904,8.078,149.514
C01832=1129.805,106.499,-56.425,-179.902,8.082,149.514
C01833=1129.800,106.749,-56.444,-179.899,8.086,149.514
C01834=1129.795,106.998,-56.462,-179.897,8.090,149.514
C01835=1129.790,107.248,-56.482,-179.894,8.094,149.515
C01836=1129.786,107.496,-56.501,-179.892,8.098,149.515
C01837=1129.781,107.746,-56.520,-179.889,8.102,149.515
C01838=1129.776,107.995,-56.538,-179.887,8.106,149.515
C01839=1129.771,108.245,-56.558,-179.885,8.110,149.516
C01840=1129.766,108.493,-56.577,-179.882,8.114,149.516
C01841=1129.762,108.743,-56.596,-179.879,8.118,149.516
C01842=1129.756,108.992,-56.615,-179.877,8.122,149.516
C01843=1129.752,109.241,-56.634,-179.875,8.126,149.516
C01844=1129.747,109.490,-56.653,-179.872,8.130,149.517
C01845=1129.742,109.740,-56.673,-179.869,8.133,149.517
C01846=1129.738,109.988,-56.692,-179.867,8.138,149.517
C01847=1129.733,110.239,-56.711,-179.865,8.141,149.517
C01848=1129.727,110.488,-56.730,-179.862,8.146,149.517
C01849=1129.723,110.737,-56.749,-179.859,8.150,149.518
C01850=1129.718,110.986,-56.768,-179.857,8.153,149.518
C01851=1129.713,111.235,-56.788,-179.855,8.157,149.518
